			(*
			ADSLOGDINT(msgCtrlMask := ADSLOG_MSGTYPE_MSGBOX OR ADSLOG_MSGTYPE_LOG,
						msgFmtStr := 'Tool life time of (T) %d actualized !',
						dintArg := BasicToolId);
			*)
		ELSE
			RRes.RESULT := WZV_TOOL_ID_BASIC_INVALID;
		END_IF
	ELSE
		(* Unknown indexgroup, just send an response *)
		RRes.LEN			:= 0;
		RRes.DATAADDR	:= 0;
		RRes.RESULT		:= ADS_RDWRT_IND_UNKNOWN_INDEXGROUP;
	END_IF
END_IF


RRes(RESPOND:=bRes);

IF bRes THEN
	RRes(RESPOND:=FALSE);
	RInd(CLEAR:=TRUE);
	RInd(CLEAR:=FALSE);
END_IF
END_METHOD

END_FUNCTION_BLOCK

// ---- POUs/CNC/F1_Init/HLI_UserInitialisation.TcPOU
FUNCTION HLI_UserInitialisation : bool
VAR_INPUT
END_VAR
VAR
END_VAR

(* ========================================================= *)
(*    FUN: HLI_UserInitialisation                            *)
(* --------------------------------------------------------- *)
(*   Desc:                                                   *)
(* Author: MK                                                *)
(*   Date: 21.12.2011                                        *)
(*   Rev.: 1.0                                               *)
(* ========================================================= *)


(* please do reset the plc program, if you change something in this module
	or in modules are in the sublevel *)

(* Axes spezific control units *)
HLI_AxisSetControlToPlc();

(* Channel 1, channel specific control unit *)
HLI_ChannelSetControlToPlc(nChan:=1);

(* Channel 2, channel specific control unit *)
HLI_ChannelSetControlToPlc(nChan:=2);

HLI_UserInitialisation := TRUE;

END_FUNCTION

// ---- POUs/CNC/F1_Init/HLI_AxisSetControlToPlc.TcPOU
FUNCTION HLI_AxisSetControlToPlc : bool
VAR_INPUT
END_VAR
VAR
 	idx						: UDINT;
END_VAR

(* ========================================================= *)
(*    FUN: HLI_AxisSetControlToPlc                           *)
(* --------------------------------------------------------- *)
(*   Desc:                                                   *)
(* Author: MK                                                *)
(*   Date: 21.12.2011                                        *)
(*   Rev.: 1.0                                               *)
(* ========================================================= *)


(* enable control units used by the program *)
FOR idx := 0 TO gNrAx - 1 DO

	IF gpAx[idx] <> 0 THEN						// check for zero pointer
		// PLC_Present for all axis
		gpAx[idx]^.head.plc_present_w := TRUE;

		// declare axis for reset
		(*gpAx[idx]^.LcControlIpo_Data.LCControlBoolUnit_PLCReset.X_Enable := TRUE;*)
		(*gpAx[idx]^.McControlIpo_Data.MCControlBoolUnit_SpdlReset.X_Enable := TRUE;*)

		(* declare axis for reference *)
		gpAx[idx]^.lr_mc_control.reference_cam.enable_w := TRUE;

		(* enable signals for real drives *)
		gpAx[idx]^.lr_mc_control.torque_permission.enable_w := TRUE;
		gpAx[idx]^.lr_mc_control.release_feedhold.enable_w := TRUE;
		gpAx[idx]^.lr_mc_control.drive_on.enable_w := TRUE;
		
		(* enable external commanding of an axis *)
		gpAx[idx]^.lr_mc_control.add_cmd_values.enable_w := TRUE;

		(* enable the axis to tracking operation (follow up) *)
		gpAx[idx]^.lr_mc_control.follow_up.enable_w := TRUE;
	END_IF

END_FOR

HLI_AxisSetControlToPlc := TRUE;

END_FUNCTION

// ---- POUs/CNC/F1_Init/HLI_ChannelSetControlToPlc.TcPOU
FUNCTION HLI_ChannelSetControlToPlc : bool
VAR_INPUT
	nChan						: UINT;
END_VAR
VAR
	nHliChIdx				: UINT;
	pChannel					: pointer to HIGH_LEVEL_INTERFACE_CH;
END_VAR

(* ========================================================= *)
(*    FUN: HLI_ChannelSetControlToPlc                        *)
(* --------------------------------------------------------- *)
(*   Desc:                                                   *)
(* Author: MK                                                *)
(*   Date: 21.12.2011                                        *)
(*   Rev.: 1.0                                               *)
(* ========================================================= *)


(* enable control units used by the program *)

nHliChIdx := nChan - 1;

IF nChan <= 0 OR gNrCh < nChan OR			(* check for channel no *)
	gpCh[nHliChIdx] = 0 THEN					(* check for zero pointer *)
	HLI_ChannelSetControlToPlc := FALSE;
	RETURN; (* e x i t *)
END_IF


pChannel := gpCh[nHliChIdx];

(* PLC_Present for the channel *)
pChannel^.head.plc_present_w := TRUE;

(* reset *)
pChannel^.bahn_lc_control.plc_reset.enable_w := TRUE;
pChannel^.channel_mc_control.mode_and_state.enable_w := TRUE;

(* override *)
pChannel^.bahn_mc_control.override_feedrate.enable_w := TRUE;

(* FeedHold *)
pChannel^.bahn_mc_control.feedhold.enable_w := TRUE;

(* Single Step *)
pChannel^.bahn_mc_control.single_block.enable_w := TRUE;

(* BackwardMotion *)
pChannel^.bahn_mc_control.backward_motion.enable_w := TRUE;

(* ReducedFeed *)
pChannel^.bahn_mc_control.reduced_speed.enable_w := TRUE;

(* Channel switch "jog of path" *)
pChannel^.bahn_mc_control.suspend_axis_output.enable_w := TRUE;

(* logon for error messages *)
pChannel^.mc_error.enable_w := TRUE;

(* program block ignore *)
pChannel^.decoder_mc_control.program_block_ignore.enable_w := TRUE;

(* Syntax Check *)
pChannel^.decoder_mc_control.execution_mode.enable_w := TRUE;

(* Optional stop M01 *)
pChannel^.bahn_mc_control.m01_stop_enable.enable_w := TRUE;

(* Enable channel specific messages handling *)
pChannel^.msg_mc_control.enable_w := TRUE;

(* Enable watchdog, for real machines
Cycle time of system task is given in 100 ns.
Cycle time of CNC is given in mikro seconds.
*)
//pChannel^.head.mc_watchdog.enable_w := TRUE;
// //pChannel^.head.mc_watchdog.cycle_time_w := 2 * TwinCAT_SystemInfoVarList._TaskInfo[1].CycleTime / 10;
//pChannel^.head.mc_watchdog.cycle_time_w := 100000;		(* 100ms *)

HLI_ChannelSetControlToPlc := TRUE;

END_FUNCTION

// ---- POUs/CNC/F9_Misc/ADSLOG.TcPOU
FUNCTION ADSLOG : BOOL
VAR_INPUT
	strMsg		: STRING;
	nDINT			: DINT;
	strArg		: STRING;
	(*strArg		: STRING(1024);*)
END_VAR
VAR
END_VAR

RETURN;

IF strArg = '' THEN
	ADSLOGDINT( msgCtrlMask := ADSLOG_MSGTYPE_MSGBOX OR
										ADSLOG_MSGTYPE_LOG,
					msgFmtStr := strMsg,
					dintArg := nDINT);
ELSE
	ADSLOGSTR(	msgCtrlMask := ADSLOG_MSGTYPE_MSGBOX OR
										ADSLOG_MSGTYPE_LOG,
					msgFmtStr := strMsg,
					strArg := strArg);
END_IF

END_FUNCTION

// ---- POUs/CncPlcProgram.TcPOU
PROGRAM CncPlcProgram
VAR
	CncChannel1					: HLI_CncChannel;
	CncChannel2					: HLI_CncChannel;
	BlockSearch_Channel1		: HLI_ChannelBlockSearch;
	//BlockSearch_Channel2		: HLI_ChannelBlockSearch;
	HLI_ChannelGetMessage1	: HLI_ChannelGetMessage;
	HLI_ChannelGetMessage2	: HLI_ChannelGetMessage;
	manualModeParam			: ARRAY[0..AXIS_MANUAL_KEYUNIT_MAX] OF ST_ManualModeParam;

	nChan							: UDINT;
	nAxisIdx						: UINT;
	bEnableTracking			: BOOL;

	RT_HomingOn					: R_TRIG;

	bReferenceCam				: BOOL;

	bSuspendAxisOutputChan1 : BOOL;
	bSuspendAxisOutputChan2 : BOOL;

	val1							: UDINT;
	val2							: UDINT;
	val3							: UDINT;

	ErrorHandler				: ARRAY [1 .. HLI_SYS_AX_MAX] OF ChannelError;  (* one error handler per channel *)
	fbClearEvents				: ADSCLEAREVENTS;
	EventMode					: E_TcEventClearModes:=TCEVENTLOGIOFFS_CLEARALL;
	ClearEvent					: BOOL;
	EventFehler					: BOOL;
	bClear						: BOOL := FALSE;

	bDummy						: BOOL;
	messageChannel1			: STRING(HLI_MSG_CONTENT_STRL) := '';
	R_TrigWatchdogMessage	: R_TRIG;
	
	cncplcprogram_manualMode:BOOL;
	cncplcprogram_automaticMode:BOOL;
END_VAR

(* ========================================================= *)
(*    PRG: CncPlcProgram                                     *)
(* --------------------------------------------------------- *)
(*   Desc:                                                   *)
(* Author: MK                                                *)
(*   Date: 21.12.2011                                        *)
(*   Rev.: 1.0                                               *)
(* ========================================================= *)


(* ---------------------------------------------- *)
(* ------- PLC part for the CNC ----------------- *)
(* ---------------------------------------------- *)

BDEControlOn := TRUE;

(* Enable axis *)
//CncAxisEnable(bEnable:=PLCAxisEnable);

CncAxisEnable(bEnable:=GVL.gvl_bEnableTracking);


(* tracking operation (follow up) on / off *)
//bEnableTracking := PLCAxisEnable; //AND (HLI_ChannelGetState(nChan:=1) <> HLI_IMCM_PROCESS_ERROR);

bEnableTracking := GVL.gvl_bEnableTracking; 

FOR nAxisIdx := 1 TO UDINT_TO_UINT(gNrAx) DO
	HLI_AxisSetTrackingOperation(nAxisNr:=nAxisIdx, bPLCAxisEnable:=bEnableTracking);
END_FOR


(* ReferenceCam *)
//HLI_AxisSetReferenceCam(Axis:=1, bReferenceCam:=bReferenceCam);
//HLI_AxisSetReferenceCam(Axis:=2, bReferenceCam:=bReferenceCam);
//HLI_AxisSetReferenceCam(Axis:=3, bReferenceCam:=bReferenceCam);
(*
HLI_AxisSetReferenceCam(Axis:=1, bReferenceCam:=IOs.IO_In_X1);
HLI_AxisSetReferenceCam(Axis:=2, bReferenceCam:=IOs.IO_In_X2);
HLI_AxisSetReferenceCam(Axis:=3, bReferenceCam:=IOs.IO_In_Y);
HLI_AxisSetReferenceCam(Axis:=4, bReferenceCam:=IOs.IO_In_Z1);
HLI_AxisSetReferenceCam(Axis:=5, bReferenceCam:=IOs.IO_In_Z2);
HLI_AxisSetReferenceCam(Axis:=6, bReferenceCam:=IOs.IO_In_B);*)

HLI_AxisSetReferenceCam(Axis:=1, bReferenceCam:=IOs.IO_In_X1);
HLI_AxisSetReferenceCam(Axis:=2, bReferenceCam:=IOs.IO_In_X2);
HLI_AxisSetReferenceCam(Axis:=3, bReferenceCam:=IOs.IO_In_Y);
HLI_AxisSetReferenceCam(Axis:=4, bReferenceCam:=IOs.IO_In_Z1);
HLI_AxisSetReferenceCam(Axis:=8, bReferenceCam:=IOs.IO_In_Z2);
HLI_AxisSetReferenceCam(Axis:=5, bReferenceCam:=IOs.IO_In_B);

(* Channel Override *)
(*PLCFeedOverride := 100;*)
PLCFeedOverride := PLCFeedOverride2;
PLCFeedOverride := 100;
HLI_ChannelSetOverride(nChan:=1, nOverride:=PLCFeedOverride*10);
HLI_ChannelSetOverride(nChan:=2, nOverride:=1000);


(* Messages from the channel *)
HLI_ChannelGetMessage1(nChan:=1, bExecute:=TRUE, bShowDlg:=TRUE);

(* get variables *)
(*val1 := GetVEChannelValue(nChan:=1, nVEIndex:=0, bGlobal:=TRUE);
val2 := GetVEChannelValue(nChan:=1, nVEIndex:=1, bGlobal:=TRUE);
*)

// MK check
(*
val1 := GetVEChannelValue(nChan:=1, nVEIndex:=2, bGlobal:=TRUE);
val2 := GetVEChannelValue(nChan:=1, nVEIndex:=3, bGlobal:=TRUE);
val3 := GetVEChannelValue(nChan:=1, nVEIndex:=4, bGlobal:=TRUE);
*)

(* set variables *)
(*SetVEChannelValue(nChan:=1, nVEIndex:=0, nVal:=2234, bGlobal:=TRUE); *)


(* Common loop for cnc error handling *)
FOR nChan := 1 TO gNrCh DO
	(* Error handling *)
	ErrorHandler[nChan](ChannelNr:=UDINT_TO_UINT(nChan));

	(* Enable watchdog for real machines *)
	(*
	SetPLCAlive(nChan);
	R_TrigWatchdogMessage(CLK := (CheckCNCAlive(nChan) = 0));
	IF R_TrigWatchdogMessage.Q THEN
		ADSLOGSTR(msgCtrlMask	:= ADSLOG_MSGTYPE_ERROR OR ADSLOG_MSGTYPE_MSGBOX OR ADSLOG_MSGTYPE_LOG,
		 			 msgFmtStr		:= 'PLC detects CNC not alive: %s',
		 			 strArg			:= 'channel x');
	END_IF
	*)
END_FOR


(*fbClearEvents(NetId := "", bClear := klaus, iMode := EventMode, tTimeout := t#1s);*)
fbClearEvents.NETID := '';	(* Local Computer *)
fbClearEvents.bClear:= bClear;
fbClearEvents.iMode:= EventMode;
fbClearEvents.tTimeout:= t#10s;


(* ---------------------------------------------- *)
(* ----------- Channel 1 ------------------------ *)
(* ---------------------------------------------- *)

nChan := 1;

(*  Suspend Channel Axis ->"jog of path" *)
HLI_ChannelSetSuspendAxisOutput(nChan:=nChan, bSuspendAxis:=bSuspendAxisOutputChan1);
bSuspendAxisOutputChan1 := FALSE;


(* manual mode over PLC *)
IF PlcManualModeSelectedAxis = 0 THEN
	PlcManualModeSelectedAxis := 1;		(* default axis *)
END_IF
(*MRODRIGUES*)
(*manualModeParam[0].nOpMode := PlcManualModeOpMode;*)
manualModeParam[0].nOpMode := GVL.gvl_Manual_nOpMode;
manualModeParam[0].nLogAxisNr := PlcManualModeSelectedAxis;
manualModeParam[0].nControlElement := 1;
manualModeParam[0].nHandwheelNr := 0;
manualModeParam[0].nHandwheelIncs := PlcManualModeHandWheelIncs;
manualModeParam[0].nHandwheelRes := PlcManualModeHandWheelRes; 
manualModeParam[0].nTipSpeed := PlcManualModeSpeed;
manualModeParam[0].nJogSpeed := PlcManualModeSpeed;
manualModeParam[0].nJogDistance := PlcManualModeIncrements;
(* manual mode keypress *)
manualModeParam[0].bKeyPos := PlcManualModeRightKey;
manualModeParam[0].bKeyNeg := PlcManualModeLeftKey;
manualModeParam[0].bKeyRapid := PlcManualModeRapidFeedKey;

(*
(* manual mode over PLC *)
manualModeParam[1].nOpMode := PlcManualModeOpMode;
manualModeParam[1].nLogAxisNr := 2;		(* second axis e.g. 2 *)
manualModeParam[1].nControlElement := 2;
manualModeParam[1].nHandwheelNr := 0;
manualModeParam[1].nHandwheelIncs := PlcManualModeHandWheelIncs;
manualModeParam[1].nHandwheelRes := PlcManualModeHandWheelRes; 
manualModeParam[1].nTipSpeed := PlcManualModeSpeed;
manualModeParam[1].nJogSpeed := PlcManualModeSpeed;
manualModeParam[1].nJogDistance := PlcManualModeIncrements;
(* manual mode keypress *)
manualModeParam[1].bKeyPos := PlcManualModeRightKey;
manualModeParam[1].bKeyNeg := PlcManualModeLeftKey;
manualModeParam[1].bKeyRapid := PlcManualModeRapidFeedKey;


(* manual mode over PLC *)
manualModeParam[2].nOpMode := PlcManualModeOpMode;
manualModeParam[2].nLogAxisNr := 3;		(* second axis e.g. 3 *)
manualModeParam[2].nControlElement := 3;
manualModeParam[2].nHandwheelNr := 0;
manualModeParam[2].nHandwheelIncs := PlcManualModeHandWheelIncs;
manualModeParam[2].nHandwheelRes := PlcManualModeHandWheelRes; 
manualModeParam[2].nTipSpeed := PlcManualModeSpeed;
manualModeParam[2].nJogSpeed := PlcManualModeSpeed;
manualModeParam[2].nJogDistance := PlcManualModeIncrements;
(* manual mode keypress *)
manualModeParam[2].bKeyPos := PlcManualModeRightKey;
manualModeParam[2].bKeyNeg := PlcManualModeLeftKey;
manualModeParam[2].bKeyRapid := PlcManualModeRapidFeedKey;
*)

(* MRODRIGUES
CncChannel1(nChan					:= nChan,
				(* Operation Mode *)
				bModeStandby		:= PLCMachineMode[nChan].Standby,
				bModeAutomatic		:= PLCMachineMode[nChan].Automatic,
				bModeManual			:= PLCMachineMode[nChan].Manual,
				bModeMDI				:= PLCMachineMode[nChan].MDI,
				bModeReference		:= PLCMachineMode[nChan].Homing,

				(* Operation State *)
				bStateSelect		:= bDummy,
				bStateReady			:= bDummy,
				bStateStart			:= PLCMachineMode[nChan].Start,
				bStateStop			:= PLCMachineMode[nChan].Stop,
				bStateReset			:= PLCMachineMode[nChan].Reset,

				(* Special Functions *)
				sProgramName		:= PLCMachineMode[nChan].ProgramName,
				sMDIString			:= PLCMachineMode[nChan].MDIString,
				bBackwardMotion	:= PLCMachineMode[nChan].Backward,
				bPrgBlockIgnore	:= PLCMachineMode[nChan].PrgBlockIgnore,
				bFeedHold			:= PLCMachineMode[nChan].FeedHold,
				bSingleBlock		:= PLCMachineMode[nChan].SingleBlock,
				bDoSingleBlock		:= PLCMachineMode[nChan].DoSingleBlock,
				bM01Stop				:= PLCMachineMode[nChan].M01Stop,
				nSyntaxCheck		:= PLCMachineMode[nChan].SyntaxCheck.nType,

				(* manual mode parameter *)
				stManualModeParam := manualModeParam);
*)

cncplcprogram_manualMode:=GVL.gvl_manualMode;
cncplcprogram_automaticMode:=GVL.gvl_automaticMode;

CncChannel1(nChan					:= nChan,
				(* Operation Mode *)
				bModeStandby		:= PLCMachineMode[nChan].Standby,
				bModeAutomatic		:= PLCMachineMode[nChan].Automatic,
				bModeManual			:= PLCMachineMode[nChan].Manual,
				bModeMDI				:= PLCMachineMode[nChan].MDI,
				bModeReference		:= PLCMachineMode[nChan].Homing,

				(* Operation State *)
				bStateSelect		:= bDummy,
				bStateReady			:= bDummy,
				bStateStart			:= PLCMachineMode[nChan].Start,
				bStateStop			:= PLCMachineMode[nChan].Stop,
				bStateReset			:= PLCMachineMode[nChan].Reset,

				(* Special Functions *)
				sProgramName		:= PLCMachineMode[nChan].ProgramName,
				sMDIString			:= PLCMachineMode[nChan].MDIString,
				bBackwardMotion	:= PLCMachineMode[nChan].Backward,
				bPrgBlockIgnore	:= PLCMachineMode[nChan].PrgBlockIgnore,
				bFeedHold			:= PLCMachineMode[nChan].FeedHold,
				bSingleBlock		:= PLCMachineMode[nChan].SingleBlock,
				bDoSingleBlock		:= PLCMachineMode[nChan].DoSingleBlock,
				bM01Stop				:= PLCMachineMode[nChan].M01Stop,
				nSyntaxCheck		:= PLCMachineMode[nChan].SyntaxCheck.nType,

				(* manual mode parameter *)
				stManualModeParam := manualModeParam);

BlockSearch_Channel1(
				nChan					:= nChan,
  				bStartRead        := PLCMachineMode[nChan].BlockSearch.bStartRead,   (* Edge signal *)
   			bStartWrite       := PLCMachineMode[nChan].BlockSearch.bStartWrite,  (* Edge signal *)
				BlockSearch			:= PLCMachineMode[nChan].BlockSearch);

CNCSystem.Channel[nChan].ActDistance := BlockSearch_Channel1.coveredDistance / 10.0;
CNCSystem.Channel[nChan].ActBlockCount := BlockSearch_Channel1.actualBlockCount_AferReset;
GVL.gvl_blockcount := BlockSearch_Channel1.actualBlockCount;

(* Axis manual mode with parallel interpolation G201 *)
PRG_ManualModeG201(nChan:=nChan);


(* ---------------------------------------------- *)
(* ----------- Channel 2 ------------------------ *)
(* ---------------------------------------------- *)

nChan := 2;

(*  Suspend Channel Axis ->"jog of path" *)
HLI_ChannelSetSuspendAxisOutput(nChan:=nChan, bSuspendAxis:=bSuspendAxisOutputChan2);
bSuspendAxisOutputChan2 := FALSE;

CncChannel2(nChan					:= nChan,
				(* Operation Mode *)
				bModeStandby		:= PLCMachineMode[nChan].Standby,
				bModeAutomatic		:= PLCMachineMode[nChan].Automatic,
				bModeManual			:= PLCMachineMode[nChan].Manual,
				bModeMDI				:= PLCMachineMode[nChan].MDI,
				bModeReference		:= PLCMachineMode[nChan].Homing,

				(* Operation State *)
				bStateSelect		:= bDummy,
				bStateReady			:= bDummy,
				bStateStart			:= PLCMachineMode[nChan].Start,
				bStateStop			:= PLCMachineMode[nChan].Stop,
				bStateReset			:= PLCMachineMode[nChan].Reset,

				(* Special Functions *)
				sProgramName		:= PLCMachineMode[nChan].ProgramName,
				sMDIString			:= PLCMachineMode[nChan].MDIString,
				bBackwardMotion	:= PLCMachineMode[nChan].Backward,
				bPrgBlockIgnore	:= PLCMachineMode[nChan].PrgBlockIgnore,
				bFeedHold			:= PLCMachineMode[nChan].FeedHold,
				bSingleBlock		:= PLCMachineMode[nChan].SingleBlock,
				bDoSingleBlock		:= PLCMachineMode[nChan].DoSingleBlock,
				bM01Stop				:= PLCMachineMode[nChan].M01Stop,
				nSyntaxCheck		:= PLCMachineMode[nChan].SyntaxCheck.nType);

END_PROGRAM

// ---- POUs/CNC/F2_Operation Mode/HLI_CncChannel.TcPOU
FUNCTION_BLOCK HLI_CncChannel
VAR_INPUT
	nChan						: UDINT;			(* Number of channel *)
	sProgramName 			: STRING(255);	(* must be xxx.nc *)
	sMDIString				: STRING(300);	(* the MDI string *)
	bBackwardMotion		: BOOL;			(* static signal *)
	bFeedHold				: BOOL;			(* static signal *)
	bReducedFeed			: BOOL;			(* static signal *)
	bSingleBlock			: BOOL;			(* static signal *)
	bPrgBlockIgnore		: BOOL;			(* static signal *)
	bM01Stop					: BOOL;			(* static signal *)
	nSyntaxCheck         : DINT;			(* static signal *)
	stManualModeParam		: ARRAY[0..AXIS_MANUAL_KEYUNIT_MAX] OF ST_ManualModeParam;
END_VAR
VAR_IN_OUT
	bModeStandby			: BOOL;			(* please only a flank *)
	bModeAutomatic			: BOOL;			(* please only a flank *)
	bModeManual				: BOOL;			(* please only a flank *)
	bModeMDI					: BOOL;			(* please only a flank *)
	bModeReference			: BOOL;			(* please only a flank *)
	(*bManual2				: BOOL;*)		(* static signal *)

	bStateSelect			: BOOL;			(* please only a flank *)
	bStateReady				: BOOL;			(* please only a flank *)
	bStateStart				: BOOL;			(* please only a flank *)
	bStateStop				: BOOL;			(* please only a flank *)
	bStateReset				: BOOL;			(* please only a flank *)
	bDoSingleBlock			: BOOL;			(* please only a flank *)
END_VAR
VAR
	nHliChIdx				: UDINT;
	pUnit						: POINTER TO MC_CONTROL_MCM_MODE_STATE_UNIT;	(* Pointer to HLI Motion Control Unit *)
	pCommand					: POINTER TO HLI_PROC_TRANS_TO_MODE_STATE;	(* Pointer to HLI channel command *)
	pChannel					: POINTER TO ST_CncChannel;						(* Pointer to channel control structure *)
	ChannelMHTFunction	: HLI_QuitChannelMHTFunction;
	ChannelResetRequest	: HLI_ChannelResetRequest;
	AxisManualMode			: ARRAY[0..AXIS_MANUAL_KEYUNIT_MAX] OF HLI_AxisManualMode;
	currentMode				: DWORD;				(* Current Mode of Operation Modes;*)
	currentState			: DWORD;				(* Current State of Operation Modes;*)

	idx						: UDINT;
	keyIdx					: INT;
	RT_ManualMode			: R_TRIG;
	RT_ErrorState			: R_TRIG;
	bManualActive			: BOOL;				(* self attitude *)
	bManualBusy				: BOOL;
	bServeNextAxisManual	: BOOL;
	bEndOfManualMode		: BOOL;
	bManualModeErr			: BOOL;
	bCheckOpModeFirst		: BOOL;

	fbRTrigReset			: R_TRIG;
	bResetRequest			: BOOL;
END_VAR

(* ========================================================= *)
(*     FB: HLI_CncChannel                                    *)
(* --------------------------------------------------------- *)
(*   Desc:                                                   *)
(* Author: MK                                                *)
(*   Date: 21.12.2011                                        *)
(*   Rev.: 1.0                                               *)
(* ========================================================= *)


nHliChIdx := nChan - 1;

IF nChan <= 0 OR gNrCh < nChan OR				(* check for channel no *)
	gpCh[nHliChIdx] = 0 THEN						(* check for zero pointer *)
	RETURN; (* e x i t *)
END_IF

(* set up pointer *)
pUnit    := ADR(gpCh[nHliChIdx]^.channel_mc_control.mode_and_state);
pCommand := ADR(pUnit^.command_w);


(* ************************************* *)
(*  Reset                                *)
(* ************************************* *)

(* ************************************* *)
(*  handle reset request                 *)
(*  (implicit reset over mode switch)    *)
(*                                       *)
(*  if code is unused regular            *)
(*  reset function of cnc core is used   *)
(* ************************************* *)

fbRTrigReset(clk:=bStateReset);
IF fbRTrigReset.Q THEN
	bStateReset := FALSE;
	bResetRequest := TRUE;
END_IF

ChannelResetRequest(nChan:=nChan, bExec:=bResetRequest);
IF bResetRequest AND NOT ChannelResetRequest.bBusy THEN
	HLI_ChannelResetMFunctions(nChan:=nChan);
	bResetRequest := FALSE;
END_IF



(* ************************************* *)
(*  Motion-Control                       *)
(* ************************************* *)

(* Backward Motion *)
HLI_ChannelSetBackwardMotion(nChan:=nChan, bBackwardMotion:=bBackwardMotion);

(* Program Block Ignore *)
HLI_ChannelSetProgramBlockIgnore(nChan:=nChan, bPrgBlockIgnore:=bPrgBlockIgnore);

(* Feed Hold *)
HLI_ChannelSetFeedHold(nChan:=nChan, bFeedHold:=bFeedHold);

(* Single Step *)
HLI_ChannelSetSingleBlock(nChan:=nChan, bSingleBlock:=bSingleBlock);

(* Reduced Feed *)
HLI_ChannelSetReducedFeed(nChan:=nChan, bReducedFeed:=bReducedFeed);

(* Syntax Check *)
HLI_ChannelSetSyntaxCheck(nChan:=nChan, nSyntaxCheck:=nSyntaxCheck);

(* Optional stop M01 *)
HLI_ChannelSetOptionalM01Stop(nChan:=nChan, bM01Stop:=bM01Stop);


(* ************************************* *)
(*  MHT-Function                         *)
(* ************************************* *)

(* MHT-Function, channel *)
ChannelMHTFunction(nChan:=nChan);

(* M-Function, axis *)
FOR idx := 1 TO gNrAx DO
	HLI_QuitAxisMFunction(nAxisNr:=UDINT_TO_UINT(idx));
END_FOR


(* ************************************* *)
(*  Spindle-Function, we don't need...   *)
(* ************************************* *)

(*
(* Turn Spindle(IAxisNr := 6); *)
IF GuiTurnSpindle = TRUE THEN
	SpindleCommand(IAxisNr := 6, CmdState := 1);
	 GuiTurnSpindle := FALSE;
END_IF

(* Turn Spindle(IAxisNr := 6); *)
IF GuiStopSpindle = TRUE THEN
	SpindleCommand(IAxisNr := 6, CmdState := 2);
	 GuiStopSpindle := FALSE;
END_IF

(* ResetSpindle(IAxisNr := 6); *)
IF GuiResetSpindle = TRUE THEN
	SpindleCommand(IAxisNr := 6, CmdState := 3);
	 GuiResetSpindle := FALSE;
ELSE
	(* wait for reset is active *)
	SpindleCommand(IAxisNr := 6, CmdState := 0);
END_IF
*)


(* ************************************* *)
(*  Channel Status Info and error        *)
(* ************************************* *)

HLI_ChannelGetStatusInfo(nChan:=nChan);
HLI_ChannelGetError(nChan:=nChan);


(* ************************************* *)
(*  do single stepping                   *)
(* ************************************* *)

(* Achtung: hier noch anpassen, nur in Abhaengigkeit vom aktuellen Status den Start setzen *)
IF bDoSingleBlock THEN
	bDoSingleBlock := FALSE;
	bStateStart := TRUE; 
	GVL.gvl_bstate_start := TRUE;
END_IF


(* ************************************* *)
(*  Operation Modes                      *)
(* ************************************* *)

(* Target modes and states *)
pChannel := ADR(CncSystem.Channel[nChan]);
OpModes();

(* OperationMode Standby *)
IF pChannel^.Mode.Standby = TRUE THEN
	HLI_ChannelModeStandby(nChan:=nChan, ProgramName:=sProgramName, pUnit:=pUnit, pCommand:=pCommand, pChannel:=pChannel);
END_IF

(* OperationMode Auto *)
IF pChannel^.Mode.Auto = TRUE THEN
	HLI_ChannelModeAuto(nChan:=nChan, ProgramName:=sProgramName, pUnit:=pUnit, pCommand:=pCommand, pChannel:=pChannel);
END_IF

(* OperationMode MDI *)
IF pChannel^.Mode.MDI THEN
	(*sProgramName := PLCCncMDIString;*)
	HLI_ChannelModeMDI(nChan:=nChan, pMDIString:=ADR(sMDIString), pUnit:=pUnit, pCommand:=pCommand, pChannel:=pChannel);
END_IF

(* OperationMode Reference *)
IF pChannel^.Mode.Homing THEN
	sProgramName := '';	(* we choose the default program: rpf.nc *)
	HLI_ChannelModeReference(nChan:=nChan, sRefPosString:=sProgramName, pUnit:=pUnit, pCommand:=pCommand, pChannel:=pChannel);
END_IF

(* OperationMode Manual *)
IF pChannel^.Mode.Manual THEN
	bEndOfManualMode := FALSE;
	HLI_ChannelModeManual(nChan:=nChan, pUnit:=pUnit, pCommand:=pCommand, pChannel:=pChannel);
END_IF


(* end of manual mode *)
IF (pChannel^.Mode.Standby
	OR pChannel^.Mode.Auto
	OR pChannel^.Mode.MDI
	OR pChannel^.Mode.Homing)
THEN
	bEndOfManualMode := TRUE;
END_IF

(* operation mode manual *)
IF pChannel^.Mode.Manual OR bManualActive THEN
	bManualActive := TRUE;

	(* sequential activation of manual axes operation *)
	bManualBusy := FALSE;
	bManualModeErr := FALSE;
	bServeNextAxisManual := TRUE;
	FOR keyIdx := 0 TO AXIS_MANUAL_KEYUNIT_MAX DO
		IF bServeNextAxisManual OR bEndOfManualMode THEN
			AxisManualMode[keyIdx](nChan				:= nChan,
											sProgramName	:= '',
											bEndManual		:= bEndOfManualMode,
											ManualModeParam:= stManualModeParam[keyIdx],
											nKeyUnitIdx		:= keyIdx,
											bManualModeHMI	:= FALSE,
											bReset			:= FALSE);
		END_IF
		bManualBusy := bManualBusy OR AxisManualMode[keyIdx].Busy;
		bServeNextAxisManual := bServeNextAxisManual AND AxisManualMode[keyIdx].IsActivated;
		IF AxisManualMode[keyIdx].Err THEN
			bManualModeErr := AxisManualMode[keyIdx].Err;		(* indicator for manual mode switching error *)
		END_IF
	END_FOR
	
	IF bManualBusy = FALSE THEN
		bModeManual := FALSE;
		bManualActive := FALSE;
	END_IF
END_IF


(* Reset *)
HLI_ChannelReset(nChan:=nChan);		(* channel *)
FOR idx := 1 TO gNrAx DO				(* axis *)
	HLI_AxisReset(nChan:=nChan, nAxisNr:=UDINT_TO_UINT(idx));
END_FOR

ACTION OpModes:
(*************************************************)
(* Restore internal state at first run           *)
(* after PLC reset                               *)
(*************************************************)


bStateStart:=GVL.gvl_bstate_start;
sProgramName:=GVL.gvl_sprogramname;


IF bCheckOpModeFirst = FALSE THEN
	bCheckOpModeFirst := TRUE;
	(*MRODRIGUES*)
	(*currentMode := HLI_ChannelGetMode(nChan:=nChan);*)
	currentMode := GVL.gvl_currentMode;
	IF currentMode = HLI_IMCM_STANDBY_MODE THEN
		pChannel^.Mode.Standby := TRUE;
	END_IF
	IF currentMode = HLI_IMCM_AUTOMATIC_MODE THEN
		pChannel^.Mode.Auto := TRUE;
	END_IF
	IF currentMode = HLI_IMCM_MDI_MODE THEN
		pChannel^.Mode.MDI := TRUE;
	END_IF
	IF currentMode = HLI_IMCM_MANUAL_MODE THEN
		pChannel^.Mode.Manual := TRUE;
	END_IF
	IF currentMode = HLI_IMCM_REFERENCE_MODE THEN
		pChannel^.Mode.Homing := TRUE;
	END_IF
END_IF


(*************************************************)
(* Operation Modes                               *)
(*************************************************)

IF bModeStandby THEN
	bModeStandby := FALSE;
	pChannel^.Mode.Standby		:= TRUE;
	pChannel^.Mode.Auto			:= FALSE;
	pChannel^.Mode.MDI			:= FALSE;
	pChannel^.Mode.Manual		:= FALSE;
	pChannel^.Mode.Homing		:= FALSE;

	pChannel^.State.Selected	:= TRUE;
	pChannel^.ProcessRunning	:= FALSE;
	pChannel^.ProcessStartTime := DT#1970-01-01-00:00;		(* reset *)
	pChannel^.ProcessEndTime	:= DT#1970-01-01-00:00;		(* reset *)
END_IF

IF bModeAutomatic THEN
	bModeAutomatic := FALSE;
	pChannel^.Mode.Standby		:= FALSE;
	pChannel^.Mode.Auto			:= TRUE;
	pChannel^.Mode.MDI			:= FALSE;
	pChannel^.Mode.Manual		:= FALSE;
	pChannel^.Mode.Homing		:= FALSE;

	pChannel^.State.Selected	:= TRUE;
	pChannel^.ProcessRunning	:= FALSE;
	pChannel^.ProcessStartTime := DT#1970-01-01-00:00;		(* reset *)
	pChannel^.ProcessEndTime	:= DT#1970-01-01-00:00;		(* reset *)
END_IF

IF bModeMDI THEN
	bModeMDI := FALSE;
	pChannel^.Mode.Standby		:= FALSE;
	pChannel^.Mode.Auto			:= FALSE;
	pChannel^.Mode.MDI			:= TRUE;
	pChannel^.Mode.Manual		:= FALSE;
	pChannel^.Mode.Homing		:= FALSE;

	pChannel^.State.Selected	:= TRUE;
	pChannel^.ProcessRunning	:= FALSE;
	pChannel^.ProcessStartTime := DT#1970-01-01-00:00;		(* reset *)
	pChannel^.ProcessEndTime	:= DT#1970-01-01-00:00;		(* reset *)
END_IF

(*MRODRIGUES*)
(*IF bModeManual THEN*)
IF GVL.gvl_manualMode THEN
	bModeManual := FALSE;
	pChannel^.Mode.Standby		:= FALSE;
	pChannel^.Mode.Auto			:= FALSE;
	pChannel^.Mode.MDI			:= FALSE;
	pChannel^.Mode.Manual		:= TRUE;
	pChannel^.Mode.Homing		:= FALSE;

	(*pChannel^.State.Selected := TRUE;*)
	pChannel^.State.Start		:= TRUE;
	pChannel^.ProcessRunning	:= FALSE;
	pChannel^.ProcessStartTime := DT#1970-01-01-00:00;		(* reset *)
	pChannel^.ProcessEndTime	:= DT#1970-01-01-00:00;		(* reset *)
END_IF

IF bModeReference THEN
	bModeReference := FALSE;
	pChannel^.Mode.Standby		:= FALSE;
	pChannel^.Mode.Auto			:= FALSE;
	pChannel^.Mode.MDI			:= FALSE;
	pChannel^.Mode.Manual		:= FALSE;
	pChannel^.Mode.Homing		:= TRUE;

	(*pChannel^.State.Selected := TRUE;*)
	pChannel^.State.Start		:= TRUE;
	pChannel^.ProcessRunning	:= FALSE;
	pChannel^.ProcessStartTime := DT#1970-01-01-00:00;		(* reset *)
	pChannel^.ProcessEndTime	:= DT#1970-01-01-00:00;		(* reset *)
END_IF



(*************************************************)
(* Operation States                              *)
(*************************************************)

(*MRODRIGUES*)
(*
currentMode := HLI_ChannelGetMode(nChan:=nChan);*)
currentMode := GVL.gvl_currentMode;
(*
currentState := HLI_ChannelGetState(nChan:=nChan);*)
currentState := GVL.gvl_currentState;

RT_ErrorState(CLK:=(currentState = HLI_IMCM_PROCESS_ERROR));
IF pChannel^.ProcessRunning = TRUE
	AND (currentState = HLI_IMCM_PROCESS_READY OR RT_ErrorState.Q)
THEN
	pChannel^.ProcessRunning := FALSE;
	pChannel^.ProcessEndTime := MySystemTime.dtSystemTime;
END_IF

CASE currentMode OF
	(*-------------------------------------------------------------------*)
	HLI_IMCM_STANDBY_MODE:
		IF bStateReset THEN
			pChannel^.Mode.Standby := TRUE;
			pChannel^.State.Reset := TRUE;
		END_IF

	(*-------------------------------------------------------------------*)
	HLI_IMCM_AUTOMATIC_MODE:
	(*
		IF bStateStart THEN
			pChannel^.State.Start := TRUE;
			IF pChannel^.ProcessRunning = FALSE THEN
				pChannel^.ProcessRunning := TRUE;
				pChannel^.ProcessStartTime := MySystemTime.dtSystemTime;
				pChannel^.ProcessEndTime	:= DT#1970-01-01-00:00;		(* reset *)
			END_IF
		END_IF
		*)
		IF GVL.gvl_bstate_start THEN
			pChannel^.State.Start := TRUE;
			IF pChannel^.ProcessRunning = FALSE THEN
				pChannel^.ProcessRunning := TRUE;
				pChannel^.ProcessStartTime := MySystemTime.dtSystemTime;
				pChannel^.ProcessEndTime	:= DT#1970-01-01-00:00;		(* reset *)
			END_IF
		END_IF

		IF bStateStop AND currentState <> HLI_IMCM_PROCESS_DESELECTED THEN
			pChannel^.State.Stop := TRUE;
		END_IF

		IF bStateReady THEN
			pChannel^.State.Ready := TRUE;
		END_IF

		IF bStateReset THEN
			pChannel^.State.Reset := TRUE;
		END_IF

	(*-------------------------------------------------------------------*)
	HLI_IMCM_MDI_MODE:
	(*
		IF bStateStart THEN
			pChannel^.State.Start := TRUE;
		END_IF
		*)

		IF GVL.gvl_bstate_start THEN
			pChannel^.State.Start := TRUE;
		END_IF

		IF bStateStop AND currentState <> HLI_IMCM_PROCESS_DESELECTED THEN
			pChannel^.State.Stop := TRUE;
		END_IF

		IF bStateReady THEN
			pChannel^.State.Ready := TRUE;
		END_IF

		IF bStateSelect THEN
			pChannel^.State.Selected := TRUE;
		END_IF

		IF bStateReset THEN
			pChannel^.State.Reset := TRUE;
		END_IF

	(*-------------------------------------------------------------------*)
	HLI_IMCM_MANUAL_MODE:
		IF bStateStart THEN
			pChannel^.State.Start := TRUE;
		END_IF

		IF bStateReady THEN
			pChannel^.State.Ready := TRUE;
		END_IF

		IF bStateStop THEN
			pChannel^.State.Stop := TRUE;
		END_IF

		IF bStateReset THEN
			pChannel^.State.Reset := TRUE;
		END_IF

		(* control to manual mode active *)
		(*
		IF HLI_GetChannelMode(nChan:=nChan) = HLI_IMCM_MANUAL_MODE
			AND HLI_GetChannelState(nChan:=nChan) = HLI_IMCM_PROCESS_DESELECTED THEN
			pChannel^.Start := TRUE;
		END_IF
		*)

	(*-------------------------------------------------------------------*)
	HLI_IMCM_REFERENCE_MODE:
		IF bStateStart THEN
			pChannel^.State.Start := TRUE;
		END_IF

		IF GVL.gvl_bstate_start THEN
			pChannel^.State.Start := TRUE;
		END_IF
	

		IF bStateStop THEN
			pChannel^.State.Stop := TRUE;
		END_IF

		IF bStateReset THEN
			pChannel^.State.Reset := TRUE;
		END_IF
END_CASE


GVL.gvl_bstate_start:=FALSE;

bStateStart := FALSE;
bStateStop := FALSE;
bStateReset := FALSE;
bStateSelect := FALSE;
END_ACTION

END_FUNCTION_BLOCK

// ---- POUs/CNC/F4_MHT-Function/HLI_QuitChannelMHTFunction.TcPOU
FUNCTION_BLOCK HLI_QuitChannelMHTFunction
VAR_INPUT
	nChan					: UDINT;									(* Number of channel *)
END_VAR
VAR_OUTPUT
	bOK					: BOOL;
END_VAR
VAR
	nHliChIdx			: UDINT;
	ChannelMFunction	: HLI_DoChannelMFunction;
	ChannelTFunction	: HLI_DoChannelTFunction;
	ChannelHFunction	: HLI_DoChannelHFunction;
	pChannelData		: POINTER TO HIGH_LEVEL_INTERFACE_CH;	(* local pointer to Data of actual Channel *)
	pActTechnoUnit		: POINTER TO TECHNO_UNIT_CH;		(* local pointer to actual techno unit *)
	idx					: UINT;									(* loop variable *)
	nFuncNr				: UDINT;									(* number of M-function *)
	nArgument			: DINT;									(* additional M-function argument *)
	nToolBasicId		: UDINT;									(* basis id of a tool *)

	pMHProcess			: POINTER TO HLI_M_H_PROZESS;
	pSProcess			: POINTER TO HLI_S_PROZESS;
	pTProcess			: POINTER TO HLI_T_PROZESS;
END_VAR

(* ========================================================= *)
(*     FB: HLI_QuitChannelMHTFunction                        *)
(* --------------------------------------------------------- *)
(*   Desc:                                                   *)
(* Author: MK                                                *)
(*   Rev.: 1.3                                               *)
(*   Date: 18.07.2002                                        *)
(*       : 08.04.2005                                        *)
(*       : 13.06.2007                                        *)
(* ========================================================= *)


nHliChIdx := nChan - 1;

IF nChan <= 0 OR gNrCh < nChan OR			(* check for channel no *)
	gpCh[nHliChIdx] = 0 THEN					(* check for zero pointer *)
	bOK := FALSE;
	RETURN; (* e x i t *)
END_IF


(* get pointer to channel data *)
pChannelData := gpCh[nHliChIdx];


(*********************************************************************)
(* Technology functions

	GCW_250_HLIIntfMFkt            :  INT := 1;
	GCW_250_HLIIntfHFkt            :  INT := 2;
	GCW_250_HLIIntfSpindel         :  INT := 3;
	GCW_250_HLIIntfTool            :  INT := 4;
	GCW_250_HLIIntfAxBlock         :  INT := 5;
	GCW_250_HLIIntfVEVariable      :  INT := 6;
	GCW_250_HLIIntfVEVariable_1    :  INT := 7;
	GCW_250_HLIIntfVEVariable_2    :  INT := 8;
	GCW_250_HLIIntfUnknown         :  INT := 9;
*)
(*********************************************************************)


(*********************************************************************)
(* test if there are open synchronisations for the standard synch unit *)
(*********************************************************************)
IF pChannelData^.used_units_std_sync_r > 0 THEN
	FOR idx := 0 TO pChannelData^.used_units_std_sync_r - 1 DO
		(* get pointer to actual techno unit *)
		pActTechnoUnit := ADR(pChannelData^.techno_unit_std_sync[idx]);
	
		IF pActTechnoUnit^.please_rw = TRUE AND						(* request from CNC *)
			pActTechnoUnit^.done_w = FALSE 							(* not acknowledged *)
		THEN
			
			(* --- M-function --- *)
			IF pActTechnoUnit^.fkt_ctrl_r = HLI_INTF_M_FKT THEN
				(* Read number of M-function *)
				pMHProcess := ADR(pActTechnoUnit^.attribut_r.data[0]);
				nFuncNr    := pMHProcess^.nr;
				nArgument	:= pMHProcess^.add_nr_r;
	
				ChannelMFunction(nChan:=nChan, nFuncNr:=nFuncNr, nArg:=nArgument);
				IF ChannelMFunction.bBusy = FALSE THEN
					(* acknowledge this M-function *)
					pActTechnoUnit^.please_rw := FALSE;
					pActTechnoUnit^.done_w := TRUE;
					ADSLOG2(strMsg:='acknowledge of M-function: %d', nUDINT:=nFuncNr, strArg:='');
				END_IF
	
				bOK := TRUE;
	
			(* --- T-function --- *)
			ELSIF pActTechnoUnit^.fkt_ctrl_r = HLI_INTF_TOOL THEN
				(* Read number of T-function *)
				pTProcess    := ADR(pActTechnoUnit^.attribut_r.data[0]);
				nToolBasicId := DINT_TO_UDINT(pTProcess^.id.basic);
	
				ChannelTFunction(nChan:=nChan, nFuncNr:=nToolBasicId);
	
				(* acknowledge this T-function *)
				pActTechnoUnit^.please_rw := FALSE;
				pActTechnoUnit^.done_w := TRUE;
				ADSLOG2(strMsg:='acknowledge of T-function: %d', nUDINT:=nToolBasicId, strArg:='');
	
				bOK := TRUE;
	
			(* --- H-function --- *)
			ELSIF pActTechnoUnit^.fkt_ctrl_r = HLI_INTF_H_FKT THEN
				(* Read number of H-function *)
				pMHProcess := ADR(pActTechnoUnit^.attribut_r.data[0]);
				nFuncNr    := pMHProcess^.nr;
				nArgument	:= pMHProcess^.add_nr_r;
	
				ChannelHFunction(nChan:=nChan, nFuncNr:=nFuncNr, nArg:=nArgument);
				IF ChannelHFunction.bBusy = FALSE THEN
					(* acknowledge this H-function *)
					pActTechnoUnit^.please_rw := FALSE;
					pActTechnoUnit^.done_w := TRUE;
					ADSLOG2(strMsg:='acknowledge of H-function: %d', nUDINT:=nFuncNr, strArg:='');
				END_IF
				bOK := TRUE;
	
			(* --- Spindle-function --- *)
			ELSIF pActTechnoUnit^.fkt_ctrl_r = HLI_INTF_SPINDEL THEN
				(* Example: read number of S-function *)
				pSProcess := ADR(pActTechnoUnit^.attribut_r.data[0]);
	
				(* ADSLOGDINT( msgCtrlMask := ADSLOG_MSGTYPE_MSGBOX OR ADSLOG_MSGTYPE_LOG,
								msgFmtStr := 'Late synch : %d',
								dintArg := pSProcess^.W_MOveCmd); *)
	
				(* Spindle M-function to general M-function list *)
				ChannelMFunction(nChan:=nChan, nFuncNr:=pSProcess^.move_cmd);
				IF ChannelMFunction.bBusy = FALSE THEN
					(* acknowledge this spindle-function *)
					pActTechnoUnit^.please_rw := FALSE;
					pActTechnoUnit^.done_w := TRUE;
				END_IF
	
				bOK := TRUE;
			END_IF
	
		END_IF
	
	END_FOR
END_IF


(*********************************************************************)
(* test if there are open synchronisations for the late synch unit *)
(*********************************************************************)
FOR idx := 0 TO HLI_TU_CH_LATE_SYNC_MAXIDX DO
	(* get pointer to actual late synch techno unit *)
	pActTechnoUnit := ADR(pChannelData^.techno_unit_late_sync[idx]);

	IF pActTechnoUnit^.please_rw = TRUE AND						(* request from CNC *)
		pActTechnoUnit^.done_w = FALSE							(* not acknowledged *)
	THEN

		(* --- M-function --- *)
		IF pActTechnoUnit^.fkt_ctrl_r = HLI_INTF_M_FKT THEN
			pMHProcess := ADR(pActTechnoUnit^.attribut_r.data[1]);
			nFuncNr    := pMHProcess^.nr;

			ChannelMFunction(nChan:=nChan, nFuncNr:=nFuncNr);
			IF ChannelMFunction.bBusy = FALSE THEN
				(* acknowledge this M-function *)
				pActTechnoUnit^.please_rw := FALSE;
				pActTechnoUnit^.done_w := TRUE;
				ADSLOG2(strMsg:='acknowledge of M-function: %d', nUDINT:=nFuncNr, strArg:='');
			END_IF

			bOK := TRUE;

		(* --- spindle-function --- *)
		(*ELSIF pActTechnoUnit^.W_FktCtrl = GCW_250_HLIIntfSpindel THEN
	 		(* Example: read number of S-function *)
			pSProzess := ADR(pActTechnoUnit^.MSTHProsessChannel_Attribut.AB_Data[1]);
			ADSLOGDINT( msgCtrlMask := ADSLOG_MSGTYPE_MSGBOX OR ADSLOG_MSGTYPE_LOG,
							msgFmtStr := 'Late synch : %d',
							dintArg := pSProzess^.W_MOveCmd);
	
			ELSIF   pActTechnoUnit^.W_FktCtrl = GCW_250_HLIIntfTool THEN
				pTProzess := ADR(pActTechnoUnit^.MSTHProsessChannel_Attribut.AB_Data[1]);
				ADSLOGDINT( msgCtrlMask := ADSLOG_MSGTYPE_MSGBOX OR ADSLOG_MSGTYPE_LOG,
							msgFmtStr := 'Late tool process: %d',
							dintArg := pTProzess^.HLIToolID_Data.D_Basic);*)
			(*ELSE
				ADSLOGDINT( msgCtrlMask := ADSLOG_MSGTYPE_MSGBOX OR ADSLOG_MSGTYPE_LOG,
							msgFmtStr := 'Channel acknowledge unknown type: %d',
							dintArg := pActTechnoUnit^.W_FktCtrl);*)
		END_IF
	END_IF

END_FOR

END_FUNCTION_BLOCK

// ---- POUs/CNC/F4_MHT-Function/HLI_DoChannelMFunction.TcPOU
FUNCTION_BLOCK HLI_DoChannelMFunction
VAR_INPUT
	nChan				: UDINT;		(* Channel number *)
	nFuncNr			: UDINT;		(* Number of M-function *)
	nArg				: DINT;		(* Argument of M-Function *)
END_VAR
VAR_OUTPUT
	bBusy				: BOOL;
END_VAR
VAR
	pChannel			: POINTER TO ST_CncChannel;
END_VAR

(* ========================================================= *)
(*     FB: HLI_DoChannelMFunction                            *)
(* --------------------------------------------------------- *)
(*   Desc:                                                   *)
(* Author: MK                                                *)
(*   Rev.: 1.1                                               *)
(*   Date: 18.07.2002                                        *)
(*       : 08.04.2005                                        *)
(* ========================================================= *)


bBusy := TRUE;

IF nChan <= 0 OR gNrCh < nChan THEN			(* check for channel no *)
	RETURN; (* e x i t *)
END_IF


pChannel := ADR(CncSystem.Channel[nChan]);

(* Synch M-Functions *)
IF nFuncNr >= 0 AND nFuncNr < MAX_M_FUNCTIONS THEN
	IF pChannel^._M[nFuncNr] = FALSE THEN		(* M-Function not set *)
		pChannel^.M[nFuncNr] := TRUE;				(* set M-Function *)
		pChannel^._M[nFuncNr] := TRUE;			(* set acknowledge *)
	ELSE
		IF pChannel^.M[nFuncNr] = FALSE THEN	(* wait for quit *)
			pChannel^._M[nFuncNr] := FALSE;		(* quit the ack *)
			bBusy := FALSE;							(* quit *)
		END_IF
	END_IF
END_IF


CASE nFuncNr OF
		(*Esperar pelo aquecimento*)
	40:
		IF (Temp_Camara_set=0 OR (IOs.Temp_Camara_out<Temp_Camara_set+100 AND IOs.Temp_Camara_out>Temp_Camara_set-100)) AND 
		(Temp_Tabuleiro_set=0 OR (IOs.Temp_Tabuleiro<Temp_Tabuleiro_set+100 AND IOs.Temp_Tabuleiro>Temp_Tabuleiro_set-100))  AND
		(Temp_Extrusor_1_set=0 OR (IOs.Temp_Extrusor_1<Temp_Extrusor_1_set+10 AND IOs.Temp_Extrusor_1>Temp_Extrusor_1_set-10)) THEN
		
			pChannel^.M[nFuncNr] := FALSE;
			
		END_IF

		(*Definir temperatura câmara*)
	41: 
		Temp_Camara_set:=nArg;
		pChannel^.M[nFuncNr] := FALSE;
		
		(*Definir temperatura câmara com espera*)
	42:
		Temp_Camara_set:=nArg;
		
	IF (IOs.Temp_Camara_out<Temp_Camara_set+100 AND IOs.Temp_Camara_out>Temp_Camara_set-100) OR (Temp_Camara_set=0 AND IOs.Temp_Camara_out<3000) THEN
		pChannel^.M[nFuncNr] := FALSE;
	END_IF
	
		(*Definir temperatura tabuleiro*)
	51: 
		Temp_Tabuleiro_set:=nArg;
		pChannel^.M[nFuncNr] := FALSE;
		
		(*Definir temperatura tabuleiro com espera*)
	52:
		Temp_Tabuleiro_set:=nArg;
		
		IF Temp_Tabuleiro_set=0 THEN
			IF (IOs.Temp_Tabuleiro<IOs.Temp_Camara_in) THEN
				pChannel^.M[nFuncNr] := FALSE;
			END_IF
		ELSIF (IOs.Temp_Tabuleiro<Temp_Tabuleiro_set+100 AND IOs.Temp_Tabuleiro>Temp_Tabuleiro_set-100) THEN
				pChannel^.M[nFuncNr] := FALSE;
		END_IF
		
		(*Definir temperatura extrusor 1*)
	61: 
		Temp_Extrusor_1_set:=nArg;
		pChannel^.M[nFuncNr] := FALSE;
		
		(*Definir temperatura extrusor 1 com espera*)
	62:
		Temp_Extrusor_1_set:=nArg;
		
		IF Temp_Extrusor_1_set=0 THEN
			IF (IOs.Temp_Extrusor_1<IOs.Temp_Camara_in) THEN
				pChannel^.M[nFuncNr] := FALSE;
			END_IF
			IF (IOs.Temp_Extrusor_1<Temp_Extrusor_1_set+100 AND IOs.Temp_Extrusor_1>Temp_Extrusor_1_set-100) THEN
				pChannel^.M[nFuncNr] := FALSE;
			END_IF
		END_IF
			
END_CASE



(* MOS *)
(*
IF nFuncNr >= 23 AND nFuncNr <= 24 THEN
	bBusy := FALSE;
END_IF
*)


(* Quit M0, M1, M2, M30 *)
IF nFuncNr = 0 OR nFuncNr = 1 OR nFuncNr = 2 OR nFuncNr = 30 THEN
	pChannel^.M[nFuncNr] := FALSE;
	pChannel^._M[nFuncNr] := FALSE;
	bBusy := FALSE;
END_IF

END_FUNCTION_BLOCK

// ---- POUs/CNC/F4_MHT-Function/HLI_DoChannelTFunction.TcPOU
FUNCTION_BLOCK HLI_DoChannelTFunction
VAR_INPUT
	nChan				: UDINT;		(* Channel number *)
	nFuncNr			: UDINT;		(* Number of T-function *)
END_VAR
VAR_OUTPUT
	bBusy				: BOOL;
END_VAR
VAR
END_VAR

(* ========================================================= *)
(*     FB: HLI_DoChannelTFunction                            *)
(* --------------------------------------------------------- *)
(*   Desc:                                                   *)
(* Author: MK                                                *)
(*   Rev.: 1.1                                               *)
(*   Date: 18.07.2002                                        *)
(*       : 08.04.2005                                        *)
(* ========================================================= *)


bBusy := TRUE;

CASE nChan OF
	1:	(* cnc channel 1 -------------------------------------- *)
		CASE nFuncNr OF
			0:		bBusy := FALSE;
			1:		bBusy := FALSE;
			2:		bBusy := FALSE;
			3:		bBusy := FALSE;

			ELSE
			ADSLOGDINT( msgCtrlMask := ADSLOG_MSGTYPE_MSGBOX OR
													ADSLOG_MSGTYPE_LOG,
								msgFmtStr := 'T-Funktion (%d), Channel 1, HLI_DoChannelTFunction() not implemented!',
								dintArg := UDINT_TO_DINT(nFuncNr));
				(* Quit the M-Function *)
				bBusy := FALSE;
		END_CASE;


	2:	(* cnc channel 2 -------------------------------------- *)
		CASE nFuncNr OF
			0:		bBusy := FALSE;
			1:		bBusy := FALSE;
			2:		bBusy := FALSE;
			3:		bBusy := FALSE;


			ELSE
				ADSLOGDINT( msgCtrlMask := ADSLOG_MSGTYPE_MSGBOX OR
													ADSLOG_MSGTYPE_LOG,
								msgFmtStr := 'T-Funktion (%d), Channel 2, HLI_DoChannelTFunction() not implemented!',
								dintArg := UDINT_TO_DINT(nFuncNr));
				(* Quit the M-Function *)
				bBusy := FALSE;
		END_CASE;

ELSE
	ADSLOGDINT( msgCtrlMask := ADSLOG_MSGTYPE_MSGBOX OR
										ADSLOG_MSGTYPE_LOG,
					msgFmtStr := 'Unknown channel number (%d) in HLI_DoChannelTFunction',
					dintArg := UDINT_TO_DINT(nChan));
	bBusy := FALSE;
END_CASE;

END_FUNCTION_BLOCK

// ---- POUs/CNC/F4_MHT-Function/HLI_DoChannelHFunction.TcPOU
FUNCTION_BLOCK HLI_DoChannelHFunction
VAR_INPUT
	nChan				: UDINT;		(* Channel number *)
	nFuncNr				: UDINT;		(* Number of M-function *)
	nArg				: DINT;		(* Argument of M-Function *)
END_VAR
VAR_OUTPUT
	bBusy				: BOOL;
END_VAR
VAR
	CncHFunction			: CncHFunctions;
END_VAR

(* ========================================================= *)
(*     FB: HLI_DoChannelHFunction                            *)
(* --------------------------------------------------------- *)
(*   Desc:                                                   *)
(* Author: MK                                                *)
(*   Rev.: 1.1                                               *)
(*   Date: 18.07.2002                                        *)
(*       : 08.04.2005                                        *)
(* ========================================================= *)


bBusy := TRUE;

CASE nChan OF
	1:	(* cnc channel 1 -------------------------------------- *)
		CASE nFuncNr OF
			0:		bBusy := FALSE;
			3:		bBusy := FALSE;
			
			1,2,11,12,21,22,31,32:
				CncHFunction(nFuncNr:=nFuncNr,nArg:=nArg);
				bBusy := TRUE;
			ELSE
				ADSLOGDINT( msgCtrlMask := ADSLOG_MSGTYPE_MSGBOX OR
													ADSLOG_MSGTYPE_LOG,
								msgFmtStr := 'H-Funktion (%d), Channel 1, HLI_DoChannelHFunction() not implemented!',
								dintArg := UDINT_TO_DINT(nFuncNr));
				(* Quit the H-Function *)
				bBusy := FALSE;
		END_CASE;


	2:	(* cnc channel 2 -------------------------------------- *)
		CASE nFuncNr OF
			0:		bBusy := FALSE;
			1:		bBusy := FALSE;
			2:		bBusy := FALSE;
			3:		bBusy := FALSE;

			ELSE
				ADSLOGDINT( msgCtrlMask := ADSLOG_MSGTYPE_MSGBOX OR
													ADSLOG_MSGTYPE_LOG,
								msgFmtStr := 'H-Funktion (%d), Channel 2, HLI_DoChannelHFunction() not implemented!',
								dintArg := UDINT_TO_DINT(nFuncNr));
				(* Quit the H-Function *)
				bBusy := FALSE;
		END_CASE;

ELSE
	ADSLOGDINT( msgCtrlMask := ADSLOG_MSGTYPE_MSGBOX OR
										ADSLOG_MSGTYPE_LOG,
					msgFmtStr := 'Unknown channel number (%d) in HLI_DoChannelHFunction',
					dintArg := UDINT_TO_DINT(nChan));
	bBusy := FALSE;
END_CASE;

END_FUNCTION_BLOCK

// ---- POUs/CncHFunctions.TcPOU
FUNCTION_BLOCK CncHFunctions
VAR_INPUT
	nFuncNr				: UDINT;		(* Number of H-function *)
	nArg				: DINT;		(* Argument of H-Function *)
END_VAR
VAR
	argument52 :DINT :=0;
	argument522 :DINT :=0;
END_VAR
VAR_OUTPUT
	Busy :BOOL;
END_VAR

(* ========================================================= *)
(*    FUN: CncHFunctions                                     *)
(* --------------------------------------------------------- *)
(*   Desc:                                                   *)
(* Author: JRM                                               *)
(*   Date: 20.12.2017                                        *)
(*   Rev.: 1.0                                               *)
(* ========================================================= *)
Busy:= TRUE;

CASE nFuncNr OF
	53:
		CASE nArg OF
			0: IOs.IO_Out_Vent_Quadro1:=FALSE;
				IOs.IO_Out_Vent_Quadro2:=FALSE;
				
			1: IOs.IO_Out_Vent_Quadro1:=TRUE;
				IOs.IO_Out_Vent_Quadro2:=FALSE;
				
			2: IOs.IO_Out_Vent_Quadro1:=TRUE;
				IOs.IO_Out_Vent_Quadro2:=TRUE;
		END_CASE
		Busy:=FALSE;
	

		
END_CASE

END_FUNCTION_BLOCK

// ---- POUs/CNC/F9_Misc/ADSLOG2.TcPOU
FUNCTION ADSLOG2 : BOOL
VAR_INPUT
	strMsg		: STRING;
	nUDINT		: UDINT;
	strArg		: STRING;
	(*strArg		: STRING(1024);*)
END_VAR
VAR
END_VAR

RETURN;

IF strArg = '' THEN
	ADSLOGDINT( msgCtrlMask := ADSLOG_MSGTYPE_MSGBOX OR
										ADSLOG_MSGTYPE_LOG,
					msgFmtStr := strMsg,
					dintArg := UDINT_TO_DINT(nUDINT));
ELSE
	ADSLOGSTR(	msgCtrlMask := ADSLOG_MSGTYPE_MSGBOX OR
										ADSLOG_MSGTYPE_LOG,
					msgFmtStr := strMsg,
					strArg := strArg);
END_IF

END_FUNCTION

// ---- POUs/CNC/F3_Control/HLI_ChannelResetRequest.TcPOU
FUNCTION_BLOCK HLI_ChannelResetRequest
VAR_INPUT
	nChan				: UDINT;		(* Channel number *)
	bExec				: BOOL;
END_VAR
VAR_OUTPUT
	bBusy				: BOOL;
END_VAR
VAR
	nState			: UINT;
	actualMode		: UDINT;
	fbTON				: TON;
	fbRtrigExec		: R_TRIG;
END_VAR

(* ========================================================= *)
(*     FB: HLI_ChannelResetRequest                           *)
(* --------------------------------------------------------- *)
(*   Desc: perform a reset in channel            				 *)
(*   Author: MiB, TV, MK                                     *)
(*   Date: 16.11.2006                                        *)
(*   Last: 16.06.2010                                        *)
(*   Rev.: 1.03                                              *)
(* ========================================================= *)


fbRtrigExec(clk := bExec);
IF fbRtrigExec.Q THEN
	bBusy := TRUE;
	nState := 10;
END_IF


CASE nState OF
	0:		(* IDLE *)
		bBusy := FALSE;

	10:	(* save actual opmode *)
		actualMode := HLI_ChannelGetMode(nChan:=nChan);

		(* switch to standby *)
		PLCMachineMode[nChan].Standby := TRUE;
		fbTON(IN:=FALSE);
		nState := 30;

	30:	(* wait for mode switch *)
		fbTON(IN:= TRUE, PT:= t#1000ms);
	 	IF HLI_ChannelGetMode(nChan:=nChan) = HLI_IMCM_STANDBY_MODE THEN
			nState := 40;
		END_IF
		IF fbTON.Q THEN
			(* Timeout Error -> go on with next step *)
			nState := 40;
		END_IF

		IF nState = 40 THEN
			(* switch back to previous mode *)
			CASE actualMode OF
				HLI_IMCM_STANDBY_MODE:		PLCMachineMode[nChan].Standby := TRUE;
				HLI_IMCM_AUTOMATIC_MODE:	PLCMachineMode[nChan].Automatic:= TRUE;
				HLI_IMCM_MDI_MODE:			PLCMachineMode[nChan].MDI:= TRUE;
				HLI_IMCM_MANUAL_MODE:		PLCMachineMode[nChan].Manual:= TRUE;
				HLI_IMCM_REFERENCE_MODE:	PLCMachineMode[nChan].Homing:= TRUE;
			ELSE
				PLCMachineMode[nChan].Standby := TRUE;
			END_CASE
			fbTON(IN:=FALSE);
			nState := 50;
		END_IF

	50:	(* wait for mode switch *)
		fbTON(IN:= TRUE, PT:= t#1000ms);
	 	IF HLI_ChannelGetMode(nChan:=nChan) = actualMode THEN
			bBusy := FALSE;
			nState := 0;
		END_IF
		IF fbTON.Q THEN
			(* Timeout Error -> go on with next step *)
			bBusy := FALSE;
			nState := 0;
		END_IF
END_CASE

END_FUNCTION_BLOCK

// ---- POUs/CNC/F3_Control/HLI_ChannelGetMode.TcPOU
FUNCTION HLI_ChannelGetMode : DWORD
VAR_INPUT
	nChan					: UDINT;			(* Number of channel *)
END_VAR
VAR
	nHliChIdx			: UDINT;
END_VAR

(* ========================================================= *)
(*    FUN: HLI_ChannelGetMode                                *)
(* --------------------------------------------------------- *)
(*   Desc:                                                   *)
(* Author: MK                                                *)
(*   Date: 21.12.2011                                        *)
(*   Rev.: 1.0                                               *)
(* ========================================================= *)


nHliChIdx := nChan - 1;

IF nChan <= 0 OR gNrCh < nChan OR			(* check for channel no *)
	gpCh[nHliChIdx] = 0 THEN					(* check for zero pointer *)
	HLI_ChannelGetMode := 0;
	RETURN; (* e x i t *)
END_IF

(* if the stop button from the HMI is selected the request is set *)
HLI_ChannelGetMode := gpCh[nHliChIdx]^.channel_mc_control.mode_and_state.state_r.mode;

END_FUNCTION

// ---- POUs/CNC/F2_Operation Mode/HLI_AxisManualMode.TcPOU
FUNCTION_BLOCK HLI_AxisManualMode
VAR_INPUT
	nChan						: UDINT;			(* Number of channel *)
	sProgramName 			: STRING(255);
	bEndManual				: BOOL;
	ManualModeParam		: ST_ManualModeParam;
	nKeyUnitIdx				: INT := 0;
	bManualModeHMI			: BOOL;			(* Manual Mode from HMI *)
	bReset					: BOOL;
	bG201						: BOOL;
END_VAR
VAR_OUTPUT
	Busy						: BOOL;
	IsActivated				: BOOL;
	Err						: BOOL;
	nErrorState				: INT;
END_VAR
VAR
	nHliChIdx				: UDINT;
	TONTimeOut				: TON;
	nState					: INT := 1;
	pString					: POINTER TO STRING;

	pChannel					: POINTER TO HIGH_LEVEL_INTERFACE_CH;  		
	pModeStateUnit			: POINTER TO MC_CONTROL_MCM_MODE_STATE_UNIT;
	pModeStateUnitCmd		: POINTER TO HLI_PROC_TRANS_TO_MODE_STATE;
	pMcControlHB			: POINTER TO MC_CONTROL_HB;
	pActivation				: POINTER TO MC_CONTROL_HB_ACTIVATION_UNIT;
	pKey						: POINTER TO MC_CONTROL_HB_KEY_UNIT;
	pRapidKey				: POINTER TO MC_CONTROL_HB_RAPID_KEY_UNIT;

	RTKeyRight				: R_TRIG;
	FTKeyRight				: F_TRIG;
	RTKeyLeft				: R_TRIG;
	FTKeyLeft				: F_TRIG;

	RTRapidKey				: R_TRIG;
	FTRapidKey				: F_TRIG;

	ManualModeParamOld	: ST_ManualModeParam;
	i							: INT;
	bDeselectFirst			: BOOL := TRUE;
END_VAR

(* ========================================================= *)
(*     FB: HLI_AxisManualMode                                *)
(* --------------------------------------------------------- *)
(*   Desc: Axis manual mode                                  *)
(*   Author: MK                                              *)
(*   Date: 18.07.2002                                        *)
(*   Last: 08.04.2017                                        *)
(*   Rev.: 2.18                                              *)
(* ========================================================= *)

isActivated := GVL.gvl_manualmode_isactivated;
Busy := GVL.gvl_manualmode_busy;
nHliChIdx := nChan - 1;

IF bManualModeHMI THEN
	Busy := FALSE;
	RETURN; (* e x i t *)
END_IF

IF bEndManual AND Busy = FALSE THEN
	RETURN; (* e x i t *)
END_IF

IF nChan <= 0 OR nChan > gNrCh			(* check for channel no *)
	OR gpCh[nHliChIdx] = 0					(* check for zero pointer *)
THEN
	Busy := FALSE;
	RETURN; (* e x i t *)
END_IF

Busy := TRUE;

IF bReset THEN
	nState := 1;
	nErrorState := 0;
	Err := FALSE;
END_IF


(* setup pointers used *)
pChannel := gpCh[nHliChIdx];
pMcControlHB := ADR(pChannel^.hb_mc_control);
pRapidKey := ADR(pMcControlHB^.rapid_key);
pKey := ADR(pMcControlHB^.key[nKeyUnitIdx]);


(* clear requests from HMI *)
IF pKey^.request_semaphor_rw THEN
	pKey^.request_semaphor_rw := FALSE;
END_IF

IF pMcControlHB^.activation.request_semaphor_rw THEN
	pMcControlHB^.activation.request_semaphor_rw := FALSE;
END_IF

IF pMcControlHB^.tip_parameter.request_semaphor_rw THEN
	pMcControlHB^.tip_parameter.request_semaphor_rw := FALSE;
END_IF

IF pMcControlHB^.jog_parameter.request_semaphor_rw THEN
	pMcControlHB^.jog_parameter.request_semaphor_rw := FALSE;
END_IF


CASE nState OF
	1: (* switch to manual mode *)
		IsActivated := FALSE;

		(* enable control unit for manual mode operation *)
		IF bManualModeHMI THEN
			pKey^.enable_w := FALSE;
			pMcControlHB^.activation.enable_w := FALSE;
		ELSE
			pKey^.enable_w := TRUE;
			pMcControlHB^.activation.enable_w := TRUE;
		END_IF

		(* enable control unit for rapid key movement *)
		pRapidKey^.enable_w := TRUE;
		
		(* set up pointer *)
		pModeStateUnit := ADR(pChannel^.channel_mc_control.mode_and_state);
		pModeStateUnitCmd := ADR(pModeStateUnit^.command_w);

		ManualModeParamOld.nOpMode := ManualModeParam.nOpMode;
		ManualModeParamOld.nTipSpeed := ManualModeParam.nTipSpeed;
		ManualModeParamOld.nJogSpeed := ManualModeParam.nJogSpeed;
		ManualModeParamOld.nHandwheelRes := ManualModeParam.nHandwheelRes;
		ManualModeParamOld.nJogDistance := ManualModeParam.nJogDistance;

		(* Copy Program name *)
		pString := ADR(pModeStateUnitCmd^.parameter);
		pString^ := sProgramName;

		(* if manual mode is not active, try to activate *)
		(*
		pModeStateUnitCmd^.to_mode := HLI_IMCM_MANUAL_MODE;
		pModeStateUnitCmd^.to_state := HLI_IMCM_PROCESS_ACTIVE; (* HLI_IMCM_PROCESS_SELECTED *)
		pModeStateUnitCmd^.channel_number := nChan;
		pModeStateUnit^.command_semaphor_rw := TRUE;
		*)
		
		TONTimeOut(IN:=FALSE);
		nErrorState := 0;
		Err := FALSE;
		nState := 11;

		(* axis manual in CNC interpolation mode G201 *)
		IF bG201 = TRUE THEN
			nState := 3;
		END_IF


	11: (* wait for mode switch *)
		TONTimeOut(IN:=TRUE, PT:=T#2S);
		IF pModeStateUnit^.state_r.mode = HLI_IMCM_MANUAL_MODE AND
			pModeStateUnit^.state_r.state = HLI_IMCM_PROCESS_ACTIVE THEN	(* HLI_IMCM_PROCESS_SELECTED *)
			TONTimeOut(IN:=FALSE);
			IF bManualModeHMI THEN
				nState := 1;
				Busy := FALSE;
			ELSE
				nState := 2;
			END_IF
		END_IF

		(* error timeout *)
		IF TONTimeOut.Q = TRUE THEN
			Err := TRUE;
			nErrorState := nState;
			nState := 99;
		END_IF


	2: (* check for deselecting axis first *)
		IF bDeselectFirst = TRUE AND nKeyUnitIdx = 0 THEN
			bDeselectFirst := FALSE;
			ManualModeParamOld.nLogAxisNr := ManualModeParam.nLogAxisNr;
			
			FOR i := 0 TO HLI_CH_AX_MAXIDX DO
				IF pChannel^.bahn_state.coord_r[i].hb_display_r.operation_mode <> 0 THEN
					ManualModeParamOld.nLogAxisNr	:= pChannel^.bahn_state.coord_r[i].log_achs_nr_r;
					EXIT;
				END_IF
			END_FOR
		END_IF

		nState := 3;

		
	3: (* parametrize *)
		IF ManualModeParam.nOpMode = HLI_HB_MODE_HR THEN		(* 1 - handwheel *)
			pMcControlHB^.handwheel_incs[ManualModeParam.nHandwheelNr].command_w := ManualModeParam.nHandwheelIncs;
			pMcControlHB^.handwheel_incs[ManualModeParam.nHandwheelNr].enable_w := TRUE;
			pMcControlHB^.hr_parameter.enable_w := TRUE;
			pMcControlHB^.hr_parameter.command_w.log_achs_nr := ManualModeParam.nLogAxisNr;
			pMcControlHB^.hr_parameter.command_w.resolution := ManualModeParam.nHandwheelRes;
			pMcControlHB^.hr_parameter.command_semaphor_rw := TRUE;
		(*ELSIF ManualModeParam.nOpMode = HLI_HB_MODE_TIP THEN	*)(* 2 - tip mode (continuous) *) (*MRODRIGUES*)
		ELSIF ManualModeParam.nOpMode = GVL.gvl_Manual_nOpMode THEN
			pMcControlHB^.tip_parameter.enable_w := TRUE;
			pMcControlHB^.tip_parameter.command_w.log_achs_nr := ManualModeParam.nLogAxisNr;
			pMcControlHB^.tip_parameter.command_w.speed := ManualModeParam.nTipSpeed * 1000/60;
			pMcControlHB^.tip_parameter.command_semaphor_rw := TRUE;
		ELSIF ManualModeParam.nOpMode = HLI_HB_MODE_JOG THEN 	(* 3 - jog mode (incremental)*)
			pMcControlHB^.jog_parameter.enable_w := TRUE;
			pMcControlHB^.jog_parameter.command_w.log_achs_nr := ManualModeParam.nLogAxisNr;
			pMcControlHB^.jog_parameter.command_w.speed := ManualModeParam.nJogSpeed * 1000/60;
			pMcControlHB^.jog_parameter.command_w.distance := ManualModeParam.nJogDistance;
			pMcControlHB^.jog_parameter.command_semaphor_rw := TRUE;
		END_IF

		TONTimeOut(IN:=FALSE);
		nState := 31;

	31: (* waiting for acknowledgement *)
		TONTimeOut(IN:=TRUE, PT:=T#200S);
		IF ManualModeParam.nOpMode = HLI_HB_MODE_HR THEN		(* 1 - handwheel *)
			IF pMcControlHB^.hr_parameter.command_semaphor_rw = FALSE THEN
				TONTimeOut(IN:=FALSE);
				nState := 4;
			END_IF
		(*ELSIF ManualModeParam.nOpMode = HLI_HB_MODE_TIP THEN	*)(* 2 - tip mode (continuous) *) (*MRODRIGUES*)
		ELSIF ManualModeParam.nOpMode = GVL.gvl_Manual_nOpMode THEN
			IF pMcControlHB^.tip_parameter.command_semaphor_rw = FALSE THEN
				TONTimeOut(IN:=FALSE);
				nState := 4;
			END_IF
		ELSIF ManualModeParam.nOpMode = HLI_HB_MODE_JOG THEN 	(* 3 - jog mode (incremental)*)
			IF pMcControlHB^.jog_parameter.command_semaphor_rw = FALSE THEN
				TONTimeOut(IN:=FALSE);
				nState := 4;
			END_IF
		END_IF

		(* error timeout *)
		IF TONTimeOut.Q = TRUE THEN
			Err := TRUE;
			nErrorState := nState;
			nState := 99;
		END_IF


	4: (* activate manual operation mode for the selected axis *)
		pActivation := ADR(pMcControlHB^.activation);
		pActivation^.command_w.log_achs_nr := ManualModeParam.nLogAxisNr;
		pActivation^.command_w.control_element := ManualModeParam.nControlElement;
		pActivation^.command_w.operation_mode := ManualModeParam.nOpMode;
		pActivation^.command_semaphor_rw := TRUE;
		nState := 41;

	41: (* waiting for acknowledgement *)
		TONTimeOut(IN:=TRUE, PT:=T#2S);
		IF pActivation^.command_semaphor_rw = FALSE THEN
			TONTimeOut(IN:=FALSE);
			nState := 7;
		END_IF

		(* error timeout *)
		IF TONTimeOut.Q = TRUE THEN
			Err := TRUE;
			nErrorState := nState;
			nState := 99;
		END_IF


	7: (* finally manual mode *)
		IsActivated := TRUE;
		
		(* handwheel *)
		IF ManualModeParam.nOpMode = HLI_HB_MODE_HR THEN
			pMcControlHB^.handwheel_incs[ManualModeParam.nHandwheelNr].command_w := ManualModeParam.nHandwheelIncs;
		END_IF

		
		(* edge detection rapid traverse speed mode *)
		IF pRapidKey^.command_semaphor_rw = FALSE THEN
			RTRapidKey(CLK := ManualModeParam.bKeyRapid);
			FTRapidKey(CLK := ManualModeParam.bKeyRapid);
		END_IF

		(* rapid traverse speed mode selected *)
		IF RTRapidKey.Q THEN
			pRapidKey^.command_w.key_pressed := 1;
			pRapidKey^.command_w.log_key_nr := ManualModeParam.nControlElement;
			pRapidKey^.command_semaphor_rw := TRUE;
		END_IF

		(* rapid traverse speed mode deselected *)
		IF FTRapidKey.Q THEN
			pRapidKey^.command_w.key_pressed := 0;
			pRapidKey^.command_w.log_key_nr := ManualModeParam.nControlElement;
			pRapidKey^.command_semaphor_rw := TRUE;
		END_IF

		
		(* edge detection *)
		IF pKey^.command_semaphor_rw = FALSE THEN
			RTKeyRight(CLK := ManualModeParam.bKeyPos AND NOT ManualModeParam.bKeyNeg);
			FTKeyRight(CLK := ManualModeParam.bKeyPos AND NOT ManualModeParam.bKeyNeg);
			RTKeyLeft(CLK := NOT ManualModeParam.bKeyPos AND ManualModeParam.bKeyNeg);
			FTKeyLeft(CLK := NOT ManualModeParam.bKeyPos AND ManualModeParam.bKeyNeg);
		END_IF

		(* right key pressed *)
		IF RTKeyRight.Q = TRUE THEN
			pKey^.command_w.log_key_nr := ManualModeParam.nControlElement;
			pKey^.command_w.direction := HLI_KEY_DIR_POS;
			pKey^.command_semaphor_rw := TRUE;
		END_IF

		(* left key pressed *)
		IF RTKeyLeft.Q = TRUE THEN
			pKey^.command_w.log_key_nr := ManualModeParam.nControlElement;
			pKey^.command_w.direction := HLI_KEY_DIR_NEG;
			pKey^.command_semaphor_rw := TRUE;
		END_IF

		(* left or right key released *)
		IF FTKeyRight.Q = TRUE OR FTKeyLeft.Q = TRUE THEN
			pKey^.command_w.log_key_nr := ManualModeParam.nControlElement;
			pKey^.command_w.direction := HLI_KEY_DIR_NONE;
			pKey^.command_semaphor_rw := TRUE;
		END_IF

		
		(* end of manual mode or parametrization changed *)
		IF pKey^.command_semaphor_rw = FALSE THEN
			IF (bEndManual = TRUE)
				OR (ManualModeParam.nLogAxisNr <> ManualModeParamOld.nLogAxisNr)
				OR (ManualModeParam.nJogDistance <> ManualModeParamOld.nJogDistance)
				OR (ManualModeParam.nOpMode <> ManualModeParamOld.nOpMode)
				OR (ManualModeParam.nTipSpeed <> ManualModeParamOld.nTipSpeed)
				OR (ManualModeParam.nJogSpeed <> ManualModeParamOld.nJogSpeed)
				OR (ManualModeParam.nHandwheelRes <> ManualModeParamOld.nHandwheelRes)
			THEN
				pKey^.command_w.log_key_nr := ManualModeParam.nControlElement;
				pKey^.command_w.direction := HLI_KEY_DIR_NONE;
				pKey^.command_semaphor_rw := TRUE;
				
				pActivation^.command_w.log_achs_nr := ManualModeParamOld.nLogAxisNr;
				pActivation^.command_w.control_element := ManualModeParam.nControlElement;
				pActivation^.command_w.operation_mode := UDINT_TO_UINT(HLI_HB_MODE_NONE);
				pActivation^.command_semaphor_rw := TRUE;

				(* switch off key control unit for handwheel movement *)
				pMcControlHB^.handwheel_incs[ManualModeParam.nHandwheelNr].enable_w := FALSE;

				TONTimeOut(IN:=FALSE);
				IsActivated := FALSE;
				nState := 9;
			END_IF
		END_IF


	9: (* waiting for acknowledgement *)
		TONTimeOut(IN:=TRUE, PT:=T#2S);
		IF pKey^.command_semaphor_rw = FALSE
			AND pActivation^.command_semaphor_rw = FALSE
		THEN
			TONTimeOut(IN:=FALSE);
			ManualModeParamOld.nLogAxisNr := ManualModeParam.nLogAxisNr;
			IF bEndManual THEN
				Busy := FALSE;
			END_IF

			nState := 1;
		END_IF

		(* error timeout *)
		IF TONTimeOut.Q = TRUE THEN
			Err := TRUE;
			nErrorState := nState;
			nState := 99;
		END_IF


	99: (* error handling *)
		TONTimeOut(IN:=FALSE);
		(* end of manual mode *)
		IF bEndManual THEN
			IsActivated := FALSE;
			Busy := FALSE;
			nState := 1;
		END_IF

END_CASE

END_FUNCTION_BLOCK

// ---- POUs/CNC/F4_MHT-Function/HLI_ChannelResetMFunctions.TcPOU
FUNCTION HLI_ChannelResetMFunctions : bool
VAR_INPUT
	nChan				: UDINT;		(* Channel number *)
END_VAR
VAR
	idx				: UDINT;
END_VAR

(* ========================================================= *)
(*    FUN: HLI_ChannelResetMFunctions                        *)
(* --------------------------------------------------------- *)
(*   Desc:                                                   *)
(* Author: MK                                                *)
(*   Date: 21.12.2011                                        *)
(*   Rev.: 1.00                                              *)
(* ========================================================= *)


IF nChan <= 0 OR gNrCh < nChan THEN			(* check for channel no *)
	HLI_ChannelResetMFunctions := FALSE;
	RETURN; (* e x i t *)
END_IF

FOR idx := 1 TO MAX_M_FUNCTIONS DO
	CncSystem.Channel[nChan].M[idx] := FALSE;
	CncSystem.Channel[nChan]._M[idx] := FALSE;
END_FOR

HLI_ChannelResetMFunctions := TRUE;

END_FUNCTION

// ---- POUs/CNC/F3_Control/HLI_ChannelSetBackwardMotion.TcPOU
FUNCTION HLI_ChannelSetBackwardMotion : BOOL
VAR_INPUT
	nChan					: UDINT;			(* Number of channel *)
	bBackwardMotion	: BOOL;
END_VAR
VAR
	nHliChIdx			: UdINT;
END_VAR

(* ========================================================= *)
(*    FUN: HLI_ChannelSetBackwardMotion                      *)
(* --------------------------------------------------------- *)
(*   Desc:                                                   *)
(* Author: MK                                                *)
(*   Date: 21.12.2011                                        *)
(*   Rev.: 1.0                                               *)
(* ========================================================= *)


nHliChIdx := nChan - 1;

IF nChan <= 0 OR gNrCh < nChan OR			(* check for channel no *)
	gpCh[nHliChIdx] = 0 THEN					(* check for zero pointer *)
	HLI_ChannelSetBackwardMotion := FALSE;
	RETURN; (* e x i t *)
END_IF

gpCh[nHliChIdx]^.bahn_mc_control.backward_motion.command_w := bBackwardMotion;

HLI_ChannelSetBackwardMotion := TRUE;

END_FUNCTION

// ---- POUs/CNC/F3_Control/HLI_ChannelSetProgramBlockIgnore.TcPOU
FUNCTION HLI_ChannelSetProgramBlockIgnore : BOOL
VAR_INPUT
	nChan					: UDINT;			(* Number of channel *)
	bPrgBlockIgnore	: BOOL;
END_VAR
VAR
	nHliChIdx			: UDINT;
END_VAR

(* ========================================================= *)
(*    FUN: HLI_ChannelSetProgramBlockIgnore                  *)
(* --------------------------------------------------------- *)
(*   Desc:                                                   *)
(* Author: MK                                                *)
(*   Date: 21.12.2011                                        *)
(*   Rev.: 1.0                                               *)
(* ========================================================= *)


nHliChIdx := nChan - 1;

IF nChan <= 0 OR gNrCh < nChan OR			(* check for channel no *)
	gpCh[nHliChIdx] = 0 THEN					(* check for zero pointer *)
	HLI_ChannelSetProgramBlockIgnore := 0;
	RETURN; (* e x i t *)
END_IF

(* program block ignore *)
// MK check
gpCh[nHliChIdx]^.decoder_mc_control.program_block_ignore.command_w := BOOL_TO_UDINT(bPrgBlockIgnore);

HLI_ChannelSetProgramBlockIgnore := TRUE;

END_FUNCTION

// ---- POUs/CNC/F3_Control/HLI_ChannelSetFeedHold.TcPOU
FUNCTION HLI_ChannelSetFeedHold : BOOL
VAR_INPUT
	nChan					: UDINT;			(* Number of channel *)
	bFeedHold			: BOOL;
END_VAR
VAR
	nHliChIdx			: UdINT;
END_VAR

(* ========================================================= *)
(*    FUN: HLI_ChannelSetFeedHold                            *)
(* --------------------------------------------------------- *)
(*   Desc:                                                   *)
(* Author: MK                                                *)
(*   Date: 18.07.2002                                        *)
(*   Rev.: 1.0                                               *)
(* ========================================================= *)


nHliChIdx := nChan - 1;

IF nChan <= 0 OR gNrCh < nChan OR			(* check for channel no *)
	gpCh[nHliChIdx] = 0 THEN					(* check for zero pointer *)
	HLI_ChannelSetFeedHold := FALSE;
	RETURN; (* e x i t *)
END_IF

(* if the stop button from the HMI is selected the request is set *)
gpCh[nHliChIdx]^.bahn_mc_control.feedhold.command_w := bFeedHold OR gpCh[nHliChIdx]^.bahn_mc_control.feedhold.request_r;

HLI_ChannelSetFeedHold := TRUE;

END_FUNCTION

// ---- POUs/CNC/F3_Control/HLI_ChannelSetSingleBlock.TcPOU
FUNCTION HLI_ChannelSetSingleBlock : BOOL
VAR_INPUT
	nChan					: UDINT;			(* Number of channel *)
	bSingleBlock		: BOOL;
END_VAR
VAR
	nHliChIdx			: UdINT;
END_VAR

(* ========================================================= *)
(*    FUN: HLI_ChannelSetSingleBlock                         *)
(* --------------------------------------------------------- *)
(*   Desc:                                                   *)
(* Author: MK                                                *)
(*   Date: 21.12.2011                                        *)
(*   Rev.: 1.0                                               *)
(* ========================================================= *)


nHliChIdx := nChan - 1;

IF nChan <= 0 OR gNrCh < nChan OR			(* check for channel no *)
	gpCh[nHliChIdx] = 0 THEN					(* check for zero pointer *)
	HLI_ChannelSetSingleBlock := FALSE;
	RETURN; (* e x i t *)
END_IF

gpCh[nHliChIdx]^.bahn_mc_control.single_block.command_w := bSingleBlock;

HLI_ChannelSetSingleBlock := TRUE;

END_FUNCTION

// ---- POUs/CNC/F3_Control/HLI_ChannelSetReducedFeed.TcPOU
FUNCTION HLI_ChannelSetReducedFeed : BOOL
VAR_INPUT
	nChan					: UDINT;			(* Number of channel *)
	bReducedFeed		: BOOL;
END_VAR
VAR
	nHliChIdx			: UDINT;
END_VAR

(* ========================================================= *)
(*    FUN: HLI_ChannelSetReducedFeed                         *)
(* --------------------------------------------------------- *)
(*   Desc:                                                   *)
(* Author: MK                                                *)
(*   Date: 18.07.2002                                        *)
(*   Rev.: 1.0                                               *)
(* ========================================================= *)


nHliChIdx := nChan - 1;

IF nChan <= 0 OR gNrCh < nChan OR			(* check for channel no *)
	gpCh[nHliChIdx] = 0 THEN					(* check for zero pointer *)
	HLI_ChannelSetReducedFeed := FALSE;
	RETURN; (* e x i t *)
END_IF

gpCh[nHliChIdx]^.bahn_mc_control.reduced_speed.command_w := bReducedFeed;

HLI_ChannelSetReducedFeed := TRUE;

END_FUNCTION

// ---- POUs/CNC/F3_Control/HLI_ChannelSetSyntaxCheck.TcPOU
FUNCTION HLI_ChannelSetSyntaxCheck : bool
VAR_INPUT
	nChan					: UDINT;			(* Number of channel *)
	nSyntaxCheck		: DINT;
END_VAR
VAR
	nHliChIdx			: UdINT;
END_VAR

(* ========================================================= *)
(*    FUN: HLI_ChannelSetSyntaxCheck                         *)
(* --------------------------------------------------------- *)
(*   Desc:                                                   *)
(* Author: MK                                                *)
(*   Date: 21.12.2011                                        *)
(*   Rev.: 1.0                                               *)
(* ========================================================= *)


nHliChIdx := nChan - 1;

IF nChan <= 0 OR gNrCh < nChan OR			(* check for channel no *)
	gpCh[nHliChIdx] = 0 THEN					(* check for zero pointer *)
	HLI_ChannelSetSyntaxCheck := FALSE;
	RETURN; (* e x i t *)
END_IF

gpCh[nHliChIdx]^.decoder_mc_control.execution_mode.command_w  := nSyntaxCheck;

HLI_ChannelSetSyntaxCheck := TRUE;

END_FUNCTION

// ---- POUs/CNC/F3_Control/HLI_ChannelSetOptionalM01Stop.TcPOU
FUNCTION HLI_ChannelSetOptionalM01Stop : bool
VAR_INPUT
	nChan					: UDINT;			(* Number of channel *)
	bM01Stop				: BOOL;
END_VAR
VAR
	nHliChIdx			: UdINT;
END_VAR

(* ========================================================= *)
(*    FUN: HLI_ChannelSetOptionalM01Stop                     *)
(* --------------------------------------------------------- *)
(*   Desc:                                                   *)
(* Author: MK                                                *)
(*   Date: 21.12.2011                                        *)
(*   Rev.: 1.0                                               *)
(* ========================================================= *)


nHliChIdx := nChan - 1;

IF nChan <= 0 OR gNrCh < nChan OR			(* check for channel no *)
	gpCh[nHliChIdx] = 0 THEN					(* check for zero pointer *)
	HLI_ChannelSetOptionalM01Stop := FALSE;
	RETURN; (* e x i t *)
END_IF

gpCh[nHliChIdx]^.bahn_mc_control.m01_stop_enable.command_w := bM01Stop;

HLI_ChannelSetOptionalM01Stop := TRUE;

END_FUNCTION

// ---- POUs/CNC/F4_MHT-Function/HLI_QuitAxisMFunction.TcPOU
FUNCTION HLI_QuitAxisMFunction : BOOL
VAR_INPUT
	nAxisNr				: UINT;											(* Number of axis *)
END_VAR

VAR
	nHliAxIdx			: UINT;											(* Index of axis specific HLI area *)
	pMHProcess			: POINTER TO HLI_M_H_PROZESS;				(* Data of a M/H techno unit *)
	pSProcess			: POINTER TO HLI_S_PROZESS;				(* Data of a spindle unit *)
	pTProcess			: POINTER TO HLI_T_PROZESS;				(* Data of a techno unit *)
	pAxisData			: POINTER TO HIGH_LEVEL_INTERFACE_AX;	(* local pointer to Data of actual Axis *)
	pActTechnoUnit		: POINTER TO TECHNO_UNIT_AX;				(* local pointer to actual techno unit *)
	idx					: UINT;											(* loop variable *)
	nToolBasicId		: UDINT;											(* basis id of a tool *)
	SpdlMoveCmd			: UINT;											(* spindle movement command *)
	Revolution			: DINT;											(* SpindleRevolution *)
	pRevolution			: POINTER TO UDINT;							(* SpindleRevolution *)
	FuncNr				: UDINT;											(* Number of M-function *)
END_VAR

(* ========================================================= *)
(*    FUN: HLI_QuitAxisMFunction                             *)
(* --------------------------------------------------------- *)
(*   Desc:                                                   *)
(* Author: MK                                                *)
(*   Rev.: 1.0                                               *)
(*   Date: 21.12.2011                                        *)
(* ========================================================= *)


HLI_QuitAxisMFunction := FALSE;
nHliAxIdx := nAxisNr - 1;

IF nAxisNr <= 0 OR gNrAx < nAxisNr OR			(* check for channel no *)
	gpAx[nHliAxIdx] = 0 THEN						(* check for zero pointer *)
	HLI_QuitAxisMFunction := FALSE;
	RETURN; (* e x i t *)
END_IF


(* get pointer to Axis data *)
pAxisData := gpAx[nHliAxIdx];

(* test if there are open synchronisations  *)
IF pAxisData^.used_units_std_sync_r > 0 THEN
	FOR idx := 0 TO pAxisData^.used_units_std_sync_r - 1 DO
	
		(* get pointer to actual techno unit *)
		pActTechnoUnit := ADR(pAxisData^.techno_unit_std_sync[idx]);
	
		(* test if this M-function has to be acknowledged *)
		IF pActTechnoUnit^.please_rw = TRUE AND			(* request from CNC *)
			pActTechnoUnit^.done_w = FALSE					(* not acknowledged *)
		THEN
	
			IF pActTechnoUnit^.fkt_ctrl_r = HLI_INTF_M_FKT THEN
				(* Example: read number of M-function *)
				pMHProcess := ADR(pActTechnoUnit^.attribut_r.data[0]);
				FuncNr := pMHProcess^.nr;
				ADSLOG2(strMsg:='Axis acknowledge of M-function: %d', nUDINT:=FuncNr, strArg:='');
			ELSE
				IF pActTechnoUnit^.fkt_ctrl_r = HLI_INTF_SPINDEL THEN (* spindle-fuction *)
					pSProcess := ADR(pActTechnoUnit^.attribut_r.data[0]);
	
					(* Example: read revolution of S-function *)
					Revolution := pSProcess^.rev;
					ADSLOG(strMsg:='Spindle S-function: %d', nDINT:=Revolution, strArg:='');
	
					(* Example: read number of S-function *)
					SpdlMoveCmd := pSProcess^.move_cmd;
					ADSLOG(strMsg:='Spindle acknowledge of M-function: %d', nDINT:=SpdlMoveCmd, strArg:='');
				ELSE
					ADSLOGDINT( msgCtrlMask := ADSLOG_MSGTYPE_MSGBOX OR ADSLOG_MSGTYPE_LOG,
									msgFmtStr := 'Axis acknowledge unknown type: %d',
									dintArg := pActTechnoUnit^.fkt_ctrl_r);
				END_IF
			END_IF
	
			(* acknowledge this M-function *)
			pActTechnoUnit^.please_rw := FALSE;
			pActTechnoUnit^.done_w := TRUE;
	
			HLI_QuitAxisMFunction := TRUE;
		END_IF
	END_FOR
END_IF

END_FUNCTION

// ---- POUs/CNC/F3_Control/HLI_ChannelGetStatusInfo.TcPOU
FUNCTION HLI_ChannelGetStatusInfo : BOOL
VAR_INPUT
	nChan					: UDINT;			(* Number of channel *)
END_VAR
VAR
	pChannel				: POINTER TO ST_CNCChannel;
END_VAR

(* ========================================================= *)
(*    FUN: HLI_GetStatusInfo                                 *)
(* --------------------------------------------------------- *)
(*   Desc: Status Info from the HLI Interface                *)
(* Author: MK                                                *)
(*   Date: 18.07.2002                                        *)
(*   Rev.: 1.0                                               *)
(* ========================================================= *)


pChannel := ADR(CncSystem.Channel[nChan]);
pChannel^.ActMode := HLI_ChannelGetMode(nChan:=nChan);
pChannel^.ActState := HLI_ChannelGetState(nChan:=nChan);

(* Translate mode *)
CASE pChannel^.ActMode OF
	HLI_IMCM_MODE:							pChannel^.ActModeString := 'Mode';
	HLI_IMCM_STANDBY_MODE:				pChannel^.ActModeString := 'StandbyMode';
	HLI_IMCM_AUTOMATIC_MODE:			pChannel^.ActModeString := 'AutomaticMode';
	HLI_IMCM_MDI_MODE:					pChannel^.ActModeString := 'MDIMode';
	HLI_IMCM_MANUAL_MODE:				pChannel^.ActModeString := 'ManualMode';
	HLI_IMCM_REFERENCE_MODE:			pChannel^.ActModeString := 'ReferenceMode';
ELSE
	pChannel^.ActModeString := '---';
END_CASE;

(* Translate state *)
CASE pChannel^.ActState OF
	HLI_IMCM_PROCESS_DESELECTED:		pChannel^.ActStateString := 'Deselected';
	HLI_IMCM_PROCESS_SELECTED:			pChannel^.ActStateString := 'Selected';
	HLI_IMCM_PROCESS_READY:				pChannel^.ActStateString := 'Ready';
	HLI_IMCM_PROCESS_ACTIVE:			pChannel^.ActStateString := 'Active';
	HLI_IMCM_PROCESS_HOLD:				pChannel^.ActStateString := 'Hold';
	HLI_IMCM_PROCESS_ERROR:				pChannel^.ActStateString := 'Error';
	HLI_IMCM_PROCESS_SELECTING:		pChannel^.ActStateString := 'Selecting';
	HLI_IMCM_PROCESS_DESELECTING:		pChannel^.ActStateString := 'Deselecting';
	HLI_IMCM_PROCESS_PREPARING:		pChannel^.ActStateString := 'Preparing';
	HLI_IMCM_PROCESS_CLEARING:			pChannel^.ActStateString := 'Clearing';
	HLI_IMCM_PROCESS_STARTING:			pChannel^.ActStateString := 'Starting';
	HLI_IMCM_PROCESS_ABORTING:			pChannel^.ActStateString := 'Aborting';
	HLI_IMCM_PROCESS_STOPPING:			pChannel^.ActStateString := 'Stopping';
	HLI_IMCM_PROCESS_RESUMING:			pChannel^.ActStateString := 'Resuming';
	HLI_IMCM_PROCESS_RESETTING:		pChannel^.ActStateString := 'Resetting';
	HLI_IMCM_PROCESS_FINISHING:		pChannel^.ActStateString := 'Finishing';
ELSE
	pChannel^.ActStateString := '---';
END_CASE;

END_FUNCTION

// ---- POUs/CNC/F3_Control/HLI_ChannelGetError.TcPOU
FUNCTION HLI_ChannelGetError : BOOL
VAR_INPUT
	nChan					: UDINT;			(* Number of channel *)
END_VAR
VAR
	nHliChIdx			: UDINT;
	pChannel				: POINTER TO ST_CncChannel;
	tmpErrorMask		: HLI_ERROR_MASKE;
	pErrorMask			: POINTER TO ARRAY [0..HLI_ERR_MASK_MAXIDX] OF BYTE;
END_VAR

(* ========================================================= *)
(*    FUN: HLI_ChannelGetError                               *)
(* --------------------------------------------------------- *)
(*   Desc: Gets the channel error                            *)
(* Return: The error flag of the channel                     *)
(* Author: MK                                                *)
(*   Date: 21.12.2011                                        *)
(*   Rev.: 1.0                                               *)
(* ========================================================= *)


nHliChIdx := nChan - 1;

IF nChan <= 0 OR gNrCh < nChan OR			(* check for channel no *)
	gpCh[nHliChIdx] = 0 THEN					(* check for zero pointer *)
	HLI_ChannelGetError := TRUE;
	RETURN; (* e x i t *)
END_IF


pChannel := ADR(CncSystem.Channel[nChan]);

(* Visualisation of Mode and State *)
pChannel^.ActMode := HLI_ChannelGetMode(nChan:=nChan);
pChannel^.ActState := HLI_ChannelGetState(nChan:=nChan);


(* Error messages id *)
IF pChannel^.ActState = HLI_IMCM_PROCESS_ERROR THEN
	pChannel^.Error := TRUE;
	pChannel^.ErrorId := gpCh[nHliChIdx]^.mc_error.satz_r.kopf.error_id;
	// MK check
	pChannel^.ErrorMask := gpCh[nHliChIdx]^.mc_error.satz_r.rumpf.maske;
	pErrorMask := ADR(pChannel^.ErrorMask);
	pErrorMask^ := gpCh[nHliChIdx]^.mc_error.satz_r.rumpf.maske.err_mask;
ELSE
	pChannel^.Error := FALSE;
	pChannel^.ErrorId := 0;
	pChannel^.ErrorMask := tmpErrorMask;
END_IF

(* Quit the error message *)
(*
IF gpCh[nHliChIdx]^.mc_error.semaphor_rw
	AND pChannel^.ActState = HLI_IMCM_PROCESS_ERROR
THEN
	pChannel^.ErrorMask := gpCh[nHliChIdx]^.mc_error.satz_r.rumpf.maske;
	gpCh[nHliChIdx]^.mc_error.semaphor_rw := FALSE;
	gpCh[nHliChIdx]^.mc_error.enable_w := FALSE;
END_IF
*)

HLI_ChannelGetError := pChannel^.Error;

END_FUNCTION

// ---- POUs/CNC/F2_Operation Mode/HLI_ChannelModeStandby.TcPOU
FUNCTION HLI_ChannelModeStandby : BOOL
VAR_INPUT
	nChan					: UDINT;			(* Number of channel *)
	ProgramName 		: STRING(HLI_IMCM_MODE_STATE_PARAM_STRL);
	pUnit					: POINTER TO MC_CONTROL_MCM_MODE_STATE_UNIT;
	pCommand				: POINTER TO HLI_PROC_TRANS_TO_MODE_STATE;
	pChannel				: POINTER TO ST_CncChannel;
END_VAR
VAR
	pString				: POINTER TO STRING(HLI_IMCM_MODE_STATE_PARAM_STRL);
END_VAR

(* ========================================================= *)
(*    FUN: HLI_ChannelModeStandby                            *)
(* --------------------------------------------------------- *)
(*   Desc: switch channel to Standby mode / xxx              *)
(* Author: MK                                                *)
(*   Date: 18.07.2002                                        *)
(*   Rev.: 1.0                                               *)
(* ========================================================= *)


IF pChannel^.State.Selected THEN
	pChannel^.State.Selected := FALSE;
	pCommand^.to_mode := HLI_IMCM_STANDBY_MODE;
	pCommand^.to_state := HLI_IMCM_PROCESS_SELECTED;
	pCommand^.channel_number := nChan;
	pString := ADR(pCommand^.parameter);
	pString^ := ProgramName;
	pUnit^.command_semaphor_rw := TRUE;
	ADSLOG(strMsg:='Standby Mode selected', nDINT:=0, strArg := '');
END_IF

IF pChannel^.State.Ready THEN
	pChannel^.State.Ready := FALSE;
	pCommand^.to_mode := HLI_IMCM_STANDBY_MODE;
	pCommand^.to_state := HLI_IMCM_PROCESS_READY;
	pCommand^.channel_number := nChan;
	pString := ADR(pCommand^.parameter);
	pString^ := ProgramName;
	pUnit^.command_semaphor_rw := TRUE;
	ADSLOG(strMsg:='Standby Mode ready', nDINT:=0, strArg := '');
END_IF

IF pChannel^.State.Start THEN
	pChannel^.State.Start := FALSE;
	pCommand^.to_mode := HLI_IMCM_STANDBY_MODE;
	pCommand^.to_state := HLI_IMCM_PROCESS_ACTIVE;
	pCommand^.channel_number := nChan;
	pString := ADR(pCommand^.parameter);
	pString^ := ProgramName;
	pUnit^.command_semaphor_rw := TRUE;
	ADSLOG(strMsg:='Programm %s started', nDINT:=0, strArg:=ProgramName);
END_IF

IF pChannel^.State.Stop THEN
	pChannel^.State.Stop := FALSE;
	pCommand^.to_mode := HLI_IMCM_STANDBY_MODE;
	pCommand^.to_state := HLI_IMCM_PROCESS_HOLD;
	pCommand^.channel_number := nChan;
	pUnit^.command_semaphor_rw := TRUE;
	ADSLOG(strMsg:='Standby Mode stopped', nDINT:=0, strArg := '');
END_IF

IF pChannel^.State.Reset THEN
	pChannel^.State.Reset := FALSE;
	pCommand^.to_mode := HLI_IMCM_STANDBY_MODE;
	pCommand^.to_state := HLI_IMCM_PROCESS_DESELECTED;
	pCommand^.channel_number := nChan;
	pUnit^.command_semaphor_rw := TRUE;
	ADSLOG(strMsg:='Standby Mode resetting', nDINT:=0, strArg := '');
END_IF

HLI_ChannelModeStandby := TRUE;

END_FUNCTION

// ---- POUs/CNC/F2_Operation Mode/HLI_ChannelModeAuto.TcPOU
FUNCTION HLI_ChannelModeAuto : BOOL
VAR_INPUT
	nChan					: UDINT;			(* Number of channel *)
	ProgramName 		: STRING(HLI_IMCM_MODE_STATE_PARAM_STRL);
	pUnit					: POINTER TO MC_CONTROL_MCM_MODE_STATE_UNIT;
	pCommand				: POINTER TO HLI_PROC_TRANS_TO_MODE_STATE;
	pChannel				: POINTER TO ST_CncChannel;
END_VAR
VAR
	pString				: POINTER TO STRING(HLI_IMCM_MODE_STATE_PARAM_STRL);
END_VAR

(* ========================================================= *)
(*    FUN: HLI_ChannelModeAuto                               *)
(* --------------------------------------------------------- *)
(*   Desc: switch channel to Automatic mode / xxx            *)
(* Author: MK                                                *)
(*   Date: 18.07.2002                                        *)
(*   Rev.: 1.0                                               *)
(* ========================================================= *)


IF pChannel^.State.Selected THEN
	pChannel^.State.Selected := FALSE;
	pCommand^.to_mode := HLI_IMCM_AUTOMATIC_MODE;
	pCommand^.to_state := HLI_IMCM_PROCESS_SELECTED;
	pCommand^.channel_number := nChan;
	pString := ADR(pCommand^.parameter);
	pString^ := ProgramName;
	pUnit^.command_semaphor_rw := TRUE;
	ADSLOG(strMsg:='Automatic selected', nDINT:=0, strArg := '');
END_IF

 
IF GVL.gvl_automaticselected THEN
	pChannel^.State.Selected := FALSE;
	pCommand^.to_mode := HLI_IMCM_AUTOMATIC_MODE;
	pCommand^.to_state := HLI_IMCM_PROCESS_SELECTED;
	pCommand^.channel_number := nChan;
	pString := ADR(pCommand^.parameter);
	pString^ := ProgramName;
	pUnit^.command_semaphor_rw := TRUE;
	ADSLOG(strMsg:='Automatic selected', nDINT:=0, strArg := '');
END_IF


IF pChannel^.State.Ready THEN
	pChannel^.State.Ready := FALSE;
	pCommand^.to_mode := HLI_IMCM_AUTOMATIC_MODE;
	pCommand^.to_state := HLI_IMCM_PROCESS_READY;
	pCommand^.channel_number := nChan;
	pString := ADR(pCommand^.parameter);
	pString^ := ProgramName;
	pUnit^.command_semaphor_rw := TRUE;
	ADSLOG(strMsg:='Automatic ready', nDINT:=0, strArg := '');
END_IF

IF pChannel^.State.Start THEN
	pChannel^.State.Start := FALSE;
	pCommand^.to_mode := HLI_IMCM_AUTOMATIC_MODE;
	pCommand^.to_state := HLI_IMCM_PROCESS_ACTIVE;
	pCommand^.channel_number := nChan;
	pString := ADR(pCommand^.parameter);
	pString^ := ProgramName;
	pUnit^.command_semaphor_rw := TRUE;
	ADSLOG(strMsg:='Programm %s started', nDINT:=0, strArg:=ProgramName);
END_IF

 //IF pChannel^.State.Stop THEN
IF GVL.gvl_automaticstop THEN
	pChannel^.State.Stop := FALSE;
	pCommand^.to_mode := HLI_IMCM_AUTOMATIC_MODE;
	pCommand^.to_state := HLI_IMCM_PROCESS_HOLD;
	pCommand^.channel_number := nChan;
	pUnit^.command_semaphor_rw := TRUE;
	ADSLOG(strMsg:='Programm stopped', nDINT:=0, strArg := '');
END_IF

//IF pChannel^.State.Reset THEN
IF GVL.gvl_automaticreset THEN
	pChannel^.State.Reset := FALSE;
	pCommand^.to_mode := HLI_IMCM_AUTOMATIC_MODE;
	pCommand^.to_state := HLI_IMCM_PROCESS_DESELECTED;
	pCommand^.channel_number := nChan;
	pUnit^.command_semaphor_rw := TRUE;
	ADSLOG(strMsg:='Automatic resetting', nDINT:=0, strArg := '');
END_IF

HLI_ChannelModeAuto := TRUE;

END_FUNCTION

// ---- POUs/CNC/F2_Operation Mode/HLI_ChannelModeMDI.TcPOU
FUNCTION HLI_ChannelModeMDI : BOOL
VAR_INPUT
	nChan					: UDINT;							(* Number of channel *)
	pMDIString 			: POINTER TO STRING(HLI_IMCM_MODE_STATE_PARAM_STRL);	(* pointer to the MDI program string *)
	pUnit					: POINTER TO MC_CONTROL_MCM_MODE_STATE_UNIT;
	pCommand				: POINTER TO HLI_PROC_TRANS_TO_MODE_STATE;
	pChannel				: POINTER TO ST_CncChannel;
END_VAR
VAR
	pString				: POINTER TO STRING(HLI_IMCM_MODE_STATE_PARAM_STRL);
END_VAR

(* ========================================================= *)
(*    FUN: HLI_ChannelModeMDI                                *)
(* --------------------------------------------------------- *)
(*   Desc: switch channel to MDI mode / xxx                  *)
(* Author: MK                                                *)
(*   Date: 18.07.2002                                        *)
(*   Rev.: 1.0                                               *)
(* ========================================================= *)


IF pChannel^.State.Selected THEN
	pChannel^.State.Selected := FALSE;
	pCommand^.to_mode := HLI_IMCM_MDI_MODE;
	pCommand^.to_state := HLI_IMCM_PROCESS_SELECTED;
	pCommand^.channel_number := nChan;
	pMDIString := ADR(pCommand^.parameter);
	pUnit^.command_semaphor_rw := TRUE;
	ADSLOG(strMsg:='MDI Mode selected', nDINT:=0, strArg := '');
END_IF

IF pChannel^.State.Ready THEN
	pChannel^.State.Ready := FALSE;
	pCommand^.to_mode := HLI_IMCM_MDI_MODE;
	pCommand^.to_state := HLI_IMCM_PROCESS_READY;
	pCommand^.channel_number := nChan;
	pMDIString := ADR(pCommand^.parameter);
	pUnit^.command_semaphor_rw := TRUE;
	ADSLOG(strMsg:='MDI Mode ready', nDINT:=0, strArg := '');
END_IF

IF pChannel^.State.Start THEN
	pChannel^.State.Start := FALSE;
	pCommand^.to_mode := HLI_IMCM_MDI_MODE;
	pCommand^.to_state := HLI_IMCM_PROCESS_ACTIVE;
	pCommand^.channel_number := nChan;
	pString := ADR(pCommand^.parameter);
	pString^ := pMDIString^;
	pUnit^.command_semaphor_rw := TRUE;
	ADSLOG(strMsg:='MDI %s started', nDINT:=0, strArg:=pMDIString^);
END_IF

IF pChannel^.State.Stop THEN
	pChannel^.State.Stop := FALSE;
	pCommand^.to_mode := HLI_IMCM_MDI_MODE;
	pCommand^.to_state := HLI_IMCM_PROCESS_HOLD;
	pCommand^.channel_number := nChan;
	pUnit^.command_semaphor_rw := TRUE;
	ADSLOG(strMsg:='MDI Mode stopped', nDINT:=0, strArg := '');
END_IF

IF pChannel^.State.Reset THEN
	pChannel^.State.Reset := FALSE;
	pCommand^.to_mode := HLI_IMCM_MDI_MODE;
	pCommand^.to_state := HLI_IMCM_PROCESS_DESELECTED;
	pCommand^.channel_number := nChan;
	pUnit^.command_semaphor_rw := TRUE;
	ADSLOG(strMsg:='MDI Mode resetting', nDINT:=0, strArg := '');
END_IF

HLI_ChannelModeMDI := TRUE;

END_FUNCTION

// ---- POUs/CNC/F2_Operation Mode/HLI_ChannelModeReference.TcPOU
FUNCTION HLI_ChannelModeReference : BOOL
VAR_INPUT
	nChan					: UDINT;			(* Number of channel *)
	sRefPosString 		: STRING(HLI_IMCM_MODE_STATE_PARAM_STRL);	(* the referencing string *)
	pUnit					: POINTER TO MC_CONTROL_MCM_MODE_STATE_UNIT;
	pCommand				: POINTER TO HLI_PROC_TRANS_TO_MODE_STATE;
	pChannel				: POINTER TO ST_CncChannel;
END_VAR
VAR
	pString				: POINTER TO STRING(HLI_IMCM_MODE_STATE_PARAM_STRL);
END_VAR

(* ========================================================= *)
(*    FUN: HLI_ChannelModeReference                          *)
(* --------------------------------------------------------- *)
(*   Desc: switch channel to Reference mode / xxx            *)
(* Author: MK                                                *)
(*   Date: 18.07.2002                                        *)
(*   Rev.: 1.0                                               *)
(* ========================================================= *)


(************************************************************
	RefPosString:
	Element: parameter ( ASCII char set, length:256 character)

	Additional possibility to parametrize homing.

	If this STRING is empty, the default program
	"rpf.nc" is used.

	else by setting axis and G-code in terms of "G74
	<axis_name_1><time_1> ...
	<axis_name_2><time_2> ...
	an individual homing can be used.
*************************************************************)


IF pChannel^.State.Selected THEN
	pChannel^.State.Selected := FALSE;
	pCommand^.to_mode := HLI_IMCM_REFERENCE_MODE;
	pCommand^.to_state := HLI_IMCM_PROCESS_SELECTED;
	pCommand^.channel_number := nChan;
	pUnit^.command_semaphor_rw := TRUE;
	ADSLOG(strMsg:='Reference selected', nDINT:=0, strArg:='');
END_IF

IF pChannel^.State.Ready THEN
	pChannel^.State.Ready := FALSE;
	pCommand^.to_mode := HLI_IMCM_REFERENCE_MODE;
	pCommand^.to_state := HLI_IMCM_PROCESS_READY;
	pCommand^.channel_number := nChan;
	pString := ADR(pCommand^.parameter);
	pUnit^.command_semaphor_rw := TRUE;
	ADSLOG(strMsg:='MDI Mode ready', nDINT:=0, strArg := '');
END_IF

IF pChannel^.State.Start THEN
	pChannel^.State.Start := FALSE;
	pCommand^.to_mode := HLI_IMCM_REFERENCE_MODE;
	pCommand^.to_state := HLI_IMCM_PROCESS_ACTIVE;
	pCommand^.channel_number := nChan;
	pString := ADR(pCommand^.parameter);
	pString^ := sRefPosString;
	pUnit^.command_semaphor_rw := TRUE;
	ADSLOG(strMsg:='Programm %s reference is started', nDINT:=0, strArg:=sRefPosString);
END_IF

IF pChannel^.State.Stop THEN
	pChannel^.State.Stop := FALSE;
	pCommand^.to_mode := HLI_IMCM_REFERENCE_MODE;
	pCommand^.to_state := HLI_IMCM_PROCESS_HOLD;
	pCommand^.channel_number := nChan;
	pUnit^.command_semaphor_rw := TRUE;
	ADSLOG(strMsg:='Reference stop is selected', nDINT:=0, strArg:='');
END_IF

IF pChannel^.State.Reset THEN
	pChannel^.State.Reset := FALSE;
	pCommand^.to_mode := HLI_IMCM_REFERENCE_MODE;
	pCommand^.to_state := HLI_IMCM_PROCESS_DESELECTED;
	pCommand^.channel_number := nChan;
	pUnit^.command_semaphor_rw := TRUE;
	ADSLOG(strMsg:='Reference reset is selected', nDINT:=0, strArg:='');
END_IF

HLI_ChannelModeReference := TRUE;

END_FUNCTION

// ---- POUs/CNC/F2_Operation Mode/HLI_ChannelModeManual.TcPOU
FUNCTION HLI_ChannelModeManual : bool
VAR_INPUT
	nChan					: UDINT;			(* Number of channel *)
	pUnit					: POINTER TO MC_CONTROL_MCM_MODE_STATE_UNIT;
	pCommand				: POINTER TO HLI_PROC_TRANS_TO_MODE_STATE;
	pChannel				: POINTER TO ST_CncChannel;
END_VAR
VAR
	pString				: POINTER TO STRING;
END_VAR

(* ========================================================= *)
(*    FUN: HLI_ChannelModeManual                             *)
(* --------------------------------------------------------- *)
(*   Desc: switch channel to Manual mode / xxx               *)
(* Author: MK                                                *)
(*   Date: 18.07.2002                                        *)
(*   Rev.: 1.0                                               *)
(* ========================================================= *)


IF pChannel^.State.Selected THEN
	pChannel^.State.Selected := FALSE;
	pCommand^.to_mode := HLI_IMCM_MANUAL_MODE;
	pCommand^.to_state := HLI_IMCM_PROCESS_SELECTED;
	pCommand^.channel_number := nChan;
	pString := ADR(pCommand^.parameter);
	pString^ := '';
	pUnit^.command_semaphor_rw := TRUE;
	ADSLOG(strMsg:='Manual Mode selected', nDINT:=0, strArg := '');
END_IF

IF pChannel^.State.Ready THEN
	pChannel^.State.Ready := FALSE;
	pCommand^.to_mode := HLI_IMCM_MANUAL_MODE;
	pCommand^.to_state := HLI_IMCM_PROCESS_READY;
	pCommand^.channel_number := nChan;
	pString := ADR(pCommand^.parameter);
	pString^ := '';
	pUnit^.command_semaphor_rw := TRUE;
	ADSLOG(strMsg:='Manual Mode ready', nDINT:=0, strArg := '');
END_IF

IF pChannel^.State.Start THEN
	pChannel^.State.Start := FALSE;
	pCommand^.to_mode := HLI_IMCM_MANUAL_MODE;
	pCommand^.to_state := HLI_IMCM_PROCESS_ACTIVE;
	pCommand^.channel_number := nChan;
	pString := ADR(pCommand^.parameter);
	pString^ := '';
	pUnit^.command_semaphor_rw := TRUE;
	ADSLOG(strMsg:='Manual Mode active', nDINT:=0, strArg := '');
END_IF

IF pChannel^.State.Stop THEN
	pChannel^.State.Stop := FALSE;
	pCommand^.to_mode := HLI_IMCM_MANUAL_MODE;
	pCommand^.to_state := HLI_IMCM_PROCESS_HOLD;
	pCommand^.channel_number := nChan;
	pUnit^.command_semaphor_rw := TRUE;
	ADSLOG(strMsg:='Manual Mode stopped', nDINT:=0, strArg := '');
END_IF

IF pChannel^.State.Reset THEN
	pChannel^.State.Reset := FALSE;
	pCommand^.to_mode := HLI_IMCM_MANUAL_MODE;
	pCommand^.to_state := HLI_IMCM_PROCESS_DESELECTED;
	pCommand^.channel_number := nChan;
	pUnit^.command_semaphor_rw := TRUE;
	ADSLOG(strMsg:='Manual Mode resetting', nDINT:=0, strArg := '');
END_IF

HLI_ChannelModeManual := TRUE;

END_FUNCTION

// ---- POUs/CNC/F2_Operation Mode/HLI_ChannelReset.TcPOU
FUNCTION HLI_ChannelReset : BOOL
VAR_INPUT
	nChan				: UDINT;		(* Channel number *)
END_VAR
VAR
	pChannel			: POINTER TO HIGH_LEVEL_INTERFACE_CH;  		(* local pointer to Data of actual Channel *)
	nHliChIdx		: UDINT;
END_VAR

(* ========================================================= *)
(*    FUN: HLI_ChannelReset                                  *)
(* --------------------------------------------------------- *)
(*   Desc:                                                   *)
(* Author: MK                                                *)
(*   Date: 21.13.2011                                        *)
(*   Rev.: 1.0                                               *)
(* ========================================================= *)


HLI_ChannelReset := FALSE;
nHliChIdx := nChan - 1;

IF nChan <= 0 OR gNrCh < nChan OR			(* check for channel no *)
	gpCh[nHliChIdx] = 0 THEN					(* check for zero pointer *)
	HLI_ChannelReset := FALSE;
	RETURN; (* e x i t *)
END_IF


(* get pointer to channel data *)
pChannel := gpCh[nHliChIdx];

(* is a reset commanded *)
IF pChannel^.bahn_lc_control.plc_reset.command_r = TRUE THEN
	(* quit this reset *)
	pChannel^.bahn_lc_control.plc_reset.state_w := TRUE;
	ADSLOG2(strMsg:='Reset of channel: %d', nUDINT:=nChan, strArg:='');
	HLI_ChannelReset := TRUE;
END_IF

END_FUNCTION

// ---- POUs/CNC/F2_Operation Mode/HLI_AxisReset.TcPOU
FUNCTION HLI_AxisReset : bool
VAR_INPUT
	nChan				: UDINT;							(* Channel number *)
	nAxisNr			: UDINT;							(* Axis number *)
END_VAR
VAR
	nHliAxIdx		: UDINT;							(* Index of axis specific HLI area *)
	pAxisData		: POINTER TO HIGH_LEVEL_INTERFACE_AX;	(* local pointer to data of actual axis *)
END_VAR

(* ========================================================= *)
(*    FUN: HLI_AxisReset                                     *)
(* --------------------------------------------------------- *)
(*   Desc:                                                   *)
(* Author: MK                                                *)
(*   Date: 21.12.2011                                        *)
(*   Rev.: 1.0                                               *)
(* ========================================================= *)


HLI_AxisReset := FALSE;
nHliAxIdx := nAxisNr - 1;

IF nAxisNr <= 0 OR gNrAx < nAxisNr		(* check for axis no *)
	OR gpAx[nHliAxIdx] = 0 THEN			(* check for zero pointer *)
	HLI_AxisReset := FALSE;
	RETURN; (* e x i t *)
END_IF


